KUKA KRL program: f1_Kuka_APT221T03S21.SRC

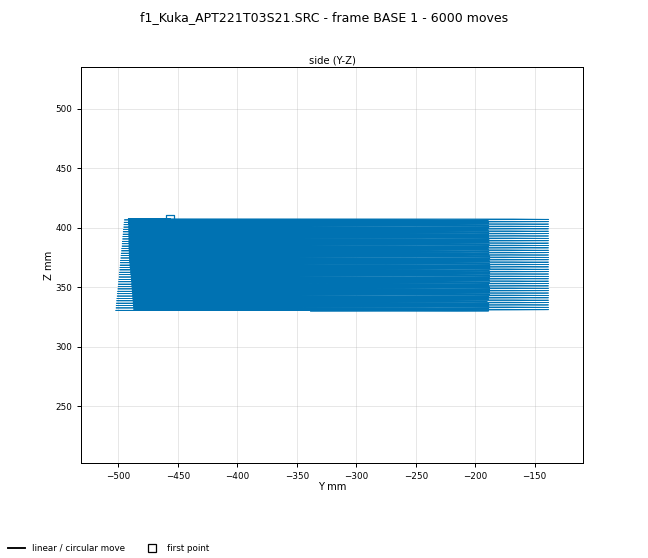
[picture p0: tool path of f1_Kuka_APT221T03S21.SRC in frame BASE 1, 6000 of 6001 moves have a stored position in this frame; points joined in program order, loops and branches not executed]
&ACCESS RVP
&REL 2
&PARAM TEMPLATE = C:\KRC\Roboter\Template\vorgabe
&PARAM EDITMASK = *
DEF f1_Kuka_APT221T03S21()


;FOLD INI;%{PE}%V3.2.0,%MKUKATPBASIS,%CINIT,%VCOMMON,%P
  ;FOLD BAS INI;%{E}%V3.2.0,%MKUKATPBASIS,%CINIT,%VINIT,%P
    GLOBAL INTERRUPT DECL 3 WHEN $STOPMESS==TRUE DO IR_STOPM ( )
    INTERRUPT ON 3
    BAS (#INITMOV,0 )
  ;ENDFOLD (BAS INI)
  ;FOLD USER INI;%{E}%V3.2.0,%MKUKATPUSER,%CINIT,%VINIT,%P
    ;Make your modifications here
  ;ENDFOLD (USER INI)
;ENDFOLD (INI)


;*** Make Null PTP Move
  PTP $pos_act

;*** Auto Load The Correct TOOL Data
  $tool=tool_data[3]

;*** Auto Load The Correct BASE Data
  $base=base_data[1]

  $ADVANCE = 5

;*** Restate Last Velocity
MMPM(30000.0)
SetRPM(6000)
LIN {X 0.057,Y -456.477,Z 407.554,A 0.000,B 0.000,C 90.000,E1 279.792} C_DIS
LIN {X 0.170,Y -464.178,Z 407.549,A 0.000,B 0.000,C 90.000,E1 278.746} C_DIS
LIN {X -0.091,Y -471.149,Z 407.543,A 0.000,B 0.000,C 90.000,E1 277.757} C_DIS
LIN {X 0.127,Y -477.448,Z 407.537,A 0.000,B 0.000,C 90.000,E1 276.720} C_DIS
LIN {X 0.133,Y -481.722,Z 407.533,A 0.000,B 0.000,C 90.000,E1 275.967} C_DIS
LIN {X 0.120,Y -485.329,Z 407.529,A 0.000,B 0.000,C 90.000,E1 275.220} C_DIS
LIN {X -0.179,Y -487.279,Z 407.526,A 0.000,B 0.000,C 90.000,E1 274.759} C_DIS
LIN {X -0.024,Y -488.832,Z 407.524,A 0.000,B 0.000,C 90.000,E1 274.245} C_DIS
LIN {X 0.180,Y -490.093,Z 407.521,A 0.000,B 0.000,C 90.000,E1 273.726} C_DIS
LIN {X -0.127,Y -490.997,Z 407.518,A 0.000,B 0.000,C 90.000,E1 273.269} C_DIS
LIN {X 0.090,Y -491.586,Z 407.515,A 0.000,B 0.000,C 90.000,E1 272.751} C_DIS
LIN {X -0.203,Y -491.810,Z 407.513,A 0.000,B 0.000,C 90.000,E1 272.293} C_DIS
LIN {X 0.017,Y -491.755,Z 407.510,A 0.000,B 0.000,C 90.000,E1 271.776} C_DIS
LIN {X 0.220,Y -491.256,Z 407.507,A 0.000,B 0.000,C 90.000,E1 271.260} C_DIS
LIN {X -0.065,Y -490.343,Z 407.504,A 0.000,B 0.000,C 90.000,E1 270.802} C_DIS
LIN {X 0.137,Y -488.944,Z 407.502,A 0.000,B 0.000,C 90.000,E1 270.286} C_DIS
LIN {X -0.154,Y -487.031,Z 407.499,A 0.000,B 0.000,C 90.000,E1 269.828} C_DIS
LIN {X 0.035,Y -484.413,Z 407.496,A 0.000,B 0.000,C 90.000,E1 269.312} C_DIS
LIN {X -0.123,Y -482.874,Z 407.495,A 0.000,B 0.000,C 90.000,E1 269.083} C_DIS
LIN {X 0.037,Y -479.075,Z 407.492,A 0.000,B 0.000,C 90.000,E1 268.568} C_DIS
LIN {X 0.188,Y -474.250,Z 407.489,A 0.000,B 0.000,C 90.000,E1 268.051} C_DIS
LIN {X 0.015,Y -471.372,Z 407.488,A 0.000,B 0.000,C 90.000,E1 267.822} C_DIS
LIN {X 0.040,Y -468.431,Z 407.487,A 0.000,B 0.000,C 90.000,E1 267.593} C_DIS
LIN {X 0.066,Y -465.066,Z 407.485,A 0.000,B 0.000,C 90.000,E1 267.364} C_DIS
LIN {X -0.070,Y -461.868,Z 407.484,A 0.000,B 0.000,C 90.000,E1 267.192} C_DIS
LIN {X -0.016,Y -454.836,Z 407.482,A 0.000,B 0.000,C 90.000,E1 266.846} C_DIS
LIN {X 0.077,Y -447.757,Z 407.481,A 0.000,B 0.000,C 90.000,E1 266.560} C_DIS
LIN {X 0.114,Y -440.498,Z 407.480,A 0.000,B 0.000,C 90.000,E1 266.331} C_DIS
LIN {X 0.063,Y -432.659,Z 407.479,A 0.000,B 0.000,C 90.000,E1 266.159} C_DIS
LIN {X -0.063,Y -423.683,Z 407.478,A 0.000,B 0.000,C 90.000,E1 266.045} C_DIS
LIN {X -0.172,Y -414.716,Z 407.478,A 0.000,B 0.000,C 90.000,E1 265.988} C_DIS
LIN {X 0.134,Y -409.225,Z 407.477,A 0.000,B 0.000,C 90.000,E1 265.927} C_DIS
LIN {X 0.029,Y -180.918,Z 407.477,A 0.000,B 0.000,C 90.000,E1 265.927} C_DIS
LIN {X 0.004,Y -180.835,Z 407.472,A 0.000,B 0.000,C 90.000,E1 264.894} C_DIS
LIN {X 0.078,Y -178.874,Z 407.443,A 0.000,B 0.000,C 90.000,E1 259.634} C_DIS
LIN {X -0.022,Y -175.916,Z 407.414,A 0.000,B 0.000,C 90.000,E1 254.574} C_DIS
LIN {X 0.034,Y -174.609,Z 407.405,A 0.000,B 0.000,C 90.000,E1 252.851} C_DIS
LIN {X -0.040,Y -171.590,Z 407.381,A 0.000,B 0.000,C 90.000,E1 248.592} C_DIS
LIN {X -0.050,Y -167.813,Z 407.357,A 0.000,B 0.000,C 90.000,E1 244.280} C_DIS
LIN {X -0.033,Y -166.534,Z 407.347,A 0.000,B 0.000,C 90.000,E1 242.538} C_DIS
LIN {X 0.017,Y -162.533,Z 407.323,A 0.000,B 0.000,C 90.000,E1 238.152} C_DIS
LIN {X -0.061,Y -161.208,Z 407.313,A 0.000,B 0.000,C 90.000,E1 236.421} C_DIS
LIN {X -0.026,Y -157.216,Z 407.289,A 0.000,B 0.000,C 90.000,E1 231.984} C_DIS
LIN {X -0.002,Y -155.943,Z 407.279,A 0.000,B 0.000,C 90.000,E1 230.194} C_DIS
LIN {X -0.043,Y -152.196,Z 407.254,A 0.000,B 0.000,C 90.000,E1 225.729} C_DIS
LIN {X -0.022,Y -150.442,Z 407.239,A 0.000,B 0.000,C 90.000,E1 223.014} C_DIS
LIN {X 0.005,Y -147.168,Z 407.214,A 0.000,B 0.000,C 90.000,E1 218.463} C_DIS
LIN {X -0.028,Y -145.184,Z 407.193,A 0.000,B 0.000,C 90.000,E1 214.818} C_DIS
LIN {X 0.008,Y -142.329,Z 407.163,A 0.000,B 0.000,C 90.000,E1 209.283} C_DIS
LIN {X 0.002,Y -141.717,Z 407.152,A 0.000,B 0.000,C 90.000,E1 207.436} C_DIS
LIN {X 0.050,Y -139.475,Z 407.116,A 0.000,B 0.000,C 90.000,E1 200.918} C_DIS
LIN {X 0.041,Y -138.972,Z 407.101,A 0.000,B 0.000,C 90.000,E1 198.127} C_DIS
LIN {X 0.030,Y -138.330,Z 407.054,A 0.000,B 0.000,C 90.000,E1 189.726} C_DIS
LIN {X 0.033,Y -139.435,Z 407.007,A 0.000,B 0.000,C 90.000,E1 181.318} C_DIS
LIN {X -0.027,Y -140.965,Z 406.976,A 0.000,B 0.000,C 90.000,E1 175.755} C_DIS
LIN {X 0.064,Y -142.720,Z 406.956,A 0.000,B 0.000,C 90.000,E1 172.008} C_DIS
LIN {X 0.022,Y -145.101,Z 406.930,A 0.000,B 0.000,C 90.000,E1 167.409} C_DIS
LIN {X 0.017,Y -147.725,Z 406.910,A 0.000,B 0.000,C 90.000,E1 163.740} C_DIS
LIN {X -0.042,Y -150.386,Z 406.889,A 0.000,B 0.000,C 90.000,E1 160.115} C_DIS
LIN {X -0.025,Y -153.817,Z 406.869,A 0.000,B 0.000,C 90.000,E1 156.485} C_DIS
LIN {X 0.035,Y -157.229,Z 406.849,A 0.000,B 0.000,C 90.000,E1 152.871} C_DIS
LIN {X -0.024,Y -161.397,Z 406.830,A 0.000,B 0.000,C 90.000,E1 149.331} C_DIS
LIN {X -0.014,Y -165.599,Z 406.810,A 0.000,B 0.000,C 90.000,E1 145.801} C_DIS
LIN {X -0.028,Y -170.523,Z 406.791,A 0.000,B 0.000,C 90.000,E1 142.316} C_DIS
LIN {X 0.015,Y -175.403,Z 406.771,A 0.000,B 0.000,C 90.000,E1 138.852} C_DIS
LIN {X 0.006,Y -181.026,Z 406.752,A 0.000,B 0.000,C 90.000,E1 135.445} C_DIS
LIN {X 0.000,Y -186.458,Z 406.734,A 0.000,B 0.000,C 90.000,E1 132.081} C_DIS
LIN {X 0.068,Y -191.082,Z 406.720,A 0.000,B 0.000,C 90.000,E1 129.564} C_DIS
LIN {X -0.005,Y -197.267,Z 406.701,A 0.000,B 0.000,C 90.000,E1 126.091} C_DIS
LIN {X -0.043,Y -296.085,Z 406.700,A 0.000,B 0.000,C 90.000,E1 126.091} C_DIS
LIN {X 0.068,Y -298.942,Z 406.700,A 0.000,B 0.000,C 90.000,E1 126.011} C_DIS
LIN {X 0.142,Y -303.617,Z 406.699,A 0.000,B 0.000,C 90.000,E1 125.724} C_DIS
LIN {X 0.039,Y -306.311,Z 406.697,A 0.000,B 0.000,C 90.000,E1 125.471} C_DIS
LIN {X 0.054,Y -310.021,Z 406.694,A 0.000,B 0.000,C 90.000,E1 124.898} C_DIS
LIN {X -0.167,Y -311.511,Z 406.692,A 0.000,B 0.000,C 90.000,E1 124.612} C_DIS
LIN {X 0.005,Y -316.928,Z 406.683,A 0.000,B 0.000,C 90.000,E1 122.959} C_DIS
LIN {X 0.033,Y -327.394,Z 406.667,A 0.000,B 0.000,C 90.000,E1 120.079} C_DIS
LIN {X 0.034,Y -339.228,Z 406.651,A 0.000,B 0.000,C 90.000,E1 117.257} C_DIS
LIN {X -0.100,Y -352.532,Z 406.636,A 0.000,B 0.000,C 90.000,E1 114.515} C_DIS
LIN {X 0.102,Y -365.691,Z 406.623,A 0.000,B 0.000,C 90.000,E1 112.078} C_DIS
LIN {X -0.112,Y -380.206,Z 406.610,A 0.000,B 0.000,C 90.000,E1 109.758} C_DIS
LIN {X -0.094,Y -396.183,Z 406.597,A 0.000,B 0.000,C 90.000,E1 107.457} C_DIS
LIN {X 0.091,Y -413.738,Z 406.584,A 0.000,B 0.000,C 90.000,E1 105.190} C_DIS
LIN {X 0.132,Y -432.973,Z 406.572,A 0.000,B 0.000,C 90.000,E1 103.008} C_DIS
LIN {X -0.111,Y -453.179,Z 406.561,A 0.000,B 0.000,C 90.000,E1 101.007} C_DIS
LIN {X -0.181,Y -473.926,Z 406.551,A 0.000,B 0.000,C 90.000,E1 99.151} C_DIS
LIN {X -0.056,Y -487.135,Z 406.545,A 0.000,B 0.000,C 90.000,E1 98.049} C_DIS
LIN {X -0.228,Y -490.973,Z 406.542,A 0.000,B 0.000,C 90.000,E1 97.644} C_DIS
LIN {X 0.151,Y -492.454,Z 406.541,A 0.000,B 0.000,C 90.000,E1 97.352} C_DIS
LIN {X -0.020,Y -493.557,Z 406.540,A 0.000,B 0.000,C 90.000,E1 97.125} C_DIS
LIN {X 0.220,Y -494.847,Z 406.537,A 0.000,B 0.000,C 90.000,E1 96.606} C_DIS
LIN {X -0.024,Y -495.105,Z 406.534,A 0.000,B 0.000,C 90.000,E1 96.144} C_DIS
LIN {X 0.229,Y -494.370,Z 406.531,A 0.000,B 0.000,C 90.000,E1 95.625} C_DIS
LIN {X -0.009,Y -492.516,Z 406.529,A 0.000,B 0.000,C 90.000,E1 95.163} C_DIS
LIN {X -0.152,Y -491.055,Z 406.527,A 0.000,B 0.000,C 90.000,E1 94.935} C_DIS
LIN {X -0.186,Y -483.507,Z 406.522,A 0.000,B 0.000,C 90.000,E1 93.955} C_DIS
LIN {X -0.221,Y -471.556,Z 406.514,A 0.000,B 0.000,C 90.000,E1 92.465} C_DIS
LIN {X -0.182,Y -454.336,Z 406.501,A 0.000,B 0.000,C 90.000,E1 90.172} C_DIS
LIN {X -0.062,Y -433.473,Z 406.483,A 0.000,B 0.000,C 90.000,E1 87.020} C_DIS
LIN {X 0.062,Y -417.355,Z 406.468,A 0.000,B 0.000,C 90.000,E1 84.318} C_DIS
LIN {X -0.032,Y -406.574,Z 406.458,A 0.000,B 0.000,C 90.000,E1 82.413} C_DIS
LIN {X -0.130,Y -392.920,Z 406.444,A 0.000,B 0.000,C 90.000,E1 79.916} C_DIS
LIN {X -0.171,Y -381.020,Z 406.431,A 0.000,B 0.000,C 90.000,E1 77.645} C_DIS
LIN {X 0.109,Y -369.476,Z 406.418,A 0.000,B 0.000,C 90.000,E1 75.283} C_DIS
LIN {X -0.142,Y -355.454,Z 406.402,A 0.000,B 0.000,C 90.000,E1 72.362} C_DIS
LIN {X -0.047,Y -343.515,Z 406.387,A 0.000,B 0.000,C 90.000,E1 69.625} C_DIS
LIN {X -0.146,Y -333.190,Z 406.373,A 0.000,B 0.000,C 90.000,E1 67.177} C_DIS
LIN {X -0.116,Y -323.180,Z 406.359,A 0.000,B 0.000,C 90.000,E1 64.665} C_DIS
LIN {X 0.012,Y -312.410,Z 406.343,A 0.000,B 0.000,C 90.000,E1 61.769} C_DIS
LIN {X -0.105,Y -301.020,Z 406.325,A 0.000,B 0.000,C 90.000,E1 58.535} C_DIS
LIN {X 0.085,Y -290.585,Z 406.307,A 0.000,B 0.000,C 90.000,E1 55.182} C_DIS
LIN {X -0.015,Y -280.969,Z 406.288,A 0.000,B 0.000,C 90.000,E1 51.823} C_DIS
LIN {X 0.086,Y -275.411,Z 406.276,A 0.000,B 0.000,C 90.000,E1 49.747} C_DIS
LIN {X 0.052,Y -269.718,Z 406.265,A 0.000,B 0.000,C 90.000,E1 47.676} C_DIS
LIN {X 0.091,Y -263.780,Z 406.253,A 0.000,B 0.000,C 90.000,E1 45.567} C_DIS
LIN {X 0.010,Y -257.732,Z 406.241,A 0.000,B 0.000,C 90.000,E1 43.461} C_DIS
LIN {X 0.017,Y -251.549,Z 406.230,A 0.000,B 0.000,C 90.000,E1 41.310} C_DIS
LIN {X 0.105,Y -243.317,Z 406.213,A 0.000,B 0.000,C 90.000,E1 38.382} C_DIS
LIN {X 0.060,Y -233.444,Z 406.193,A 0.000,B 0.000,C 90.000,E1 34.692} C_DIS
LIN {X 0.083,Y -226.277,Z 406.176,A 0.000,B 0.000,C 90.000,E1 31.671} C_DIS
LIN {X 0.060,Y -218.050,Z 406.155,A 0.000,B 0.000,C 90.000,E1 27.847} C_DIS
LIN {X -0.076,Y -212.245,Z 406.138,A 0.000,B 0.000,C 90.000,E1 24.771} C_DIS
LIN {X 0.063,Y -205.875,Z 406.116,A 0.000,B 0.000,C 90.000,E1 20.791} C_DIS
LIN {X 0.031,Y -200.411,Z 406.093,A 0.000,B 0.000,C 90.000,E1 16.804} C_DIS
LIN {X -0.002,Y -195.980,Z 406.071,A 0.000,B 0.000,C 90.000,E1 12.771} C_DIS
LIN {X 0.032,Y -192.503,Z 406.048,A 0.000,B 0.000,C 90.000,E1 8.681} C_DIS
LIN {X 0.027,Y -189.559,Z 406.016,A 0.000,B 0.000,C 90.000,E1 2.922} C_DIS
LIN {X -0.068,Y -189.023,Z 405.974,A 0.000,B 0.000,C 90.000,E1 355.412} C_DIS
LIN {X 0.078,Y -191.530,Z 405.938,A 0.000,B 0.000,C 90.000,E1 348.757} C_DIS
LIN {X -0.046,Y -194.931,Z 405.910,A 0.000,B 0.000,C 90.000,E1 343.866} C_DIS
LIN {X 0.082,Y -198.897,Z 405.888,A 0.000,B 0.000,C 90.000,E1 339.752} C_DIS
LIN {X -0.013,Y -203.955,Z 405.865,A 0.000,B 0.000,C 90.000,E1 335.741} C_DIS
LIN {X -0.089,Y -210.064,Z 405.843,A 0.000,B 0.000,C 90.000,E1 331.769} C_DIS
LIN {X 0.069,Y -216.918,Z 405.821,A 0.000,B 0.000,C 90.000,E1 327.788} C_DIS
LIN {X 0.064,Y -224.337,Z 405.800,A 0.000,B 0.000,C 90.000,E1 323.909} C_DIS
LIN {X -0.029,Y -232.586,Z 405.778,A 0.000,B 0.000,C 90.000,E1 320.114} C_DIS
LIN {X -0.032,Y -239.931,Z 405.762,A 0.000,B 0.000,C 90.000,E1 317.106} C_DIS
LIN {X -0.051,Y -249.284,Z 405.743,A 0.000,B 0.000,C 90.000,E1 313.785} C_DIS
LIN {X -0.119,Y -259.993,Z 405.725,A 0.000,B 0.000,C 90.000,E1 310.539} C_DIS
LIN {X 0.034,Y -271.763,Z 405.707,A 0.000,B 0.000,C 90.000,E1 307.317} C_DIS
LIN {X -0.002,Y -285.718,Z 405.688,A 0.000,B 0.000,C 90.000,E1 303.865} C_DIS
LIN {X 0.171,Y -300.414,Z 405.669,A 0.000,B 0.000,C 90.000,E1 300.463} C_DIS
LIN {X 0.053,Y -311.660,Z 405.657,A 0.000,B 0.000,C 90.000,E1 298.180} C_DIS
LIN {X 0.074,Y -327.714,Z 405.641,A 0.000,B 0.000,C 90.000,E1 295.283} C_DIS
LIN {X 0.151,Y -339.486,Z 405.630,A 0.000,B 0.000,C 90.000,E1 293.387} C_DIS
LIN {X -0.044,Y -358.914,Z 405.615,A 0.000,B 0.000,C 90.000,E1 290.663} C_DIS
LIN {X 0.048,Y -379.551,Z 405.600,A 0.000,B 0.000,C 90.000,E1 288.000} C_DIS
LIN {X 0.190,Y -404.938,Z 405.585,A 0.000,B 0.000,C 90.000,E1 285.190} C_DIS
LIN {X -0.153,Y -422.776,Z 405.575,A 0.000,B 0.000,C 90.000,E1 283.467} C_DIS
LIN {X 0.019,Y -435.520,Z 405.568,A 0.000,B 0.000,C 90.000,E1 282.175} C_DIS
LIN {X -0.089,Y -442.879,Z 405.563,A 0.000,B 0.000,C 90.000,E1 281.422} C_DIS
LIN {X 0.147,Y -449.870,Z 405.559,A 0.000,B 0.000,C 90.000,E1 280.602} C_DIS
LIN {X -0.085,Y -456.195,Z 405.555,A 0.000,B 0.000,C 90.000,E1 279.849} C_DIS
LIN {X -0.185,Y -462.061,Z 405.550,A 0.000,B 0.000,C 90.000,E1 279.086} C_DIS
LIN {X -0.083,Y -469.205,Z 405.545,A 0.000,B 0.000,C 90.000,E1 278.049} C_DIS
LIN {X 0.114,Y -475.706,Z 405.539,A 0.000,B 0.000,C 90.000,E1 277.011} C_DIS
LIN {X 0.103,Y -480.119,Z 405.535,A 0.000,B 0.000,C 90.000,E1 276.258} C_DIS
LIN {X 0.083,Y -483.997,Z 405.531,A 0.000,B 0.000,C 90.000,E1 275.511} C_DIS
LIN {X 0.136,Y -487.131,Z 405.527,A 0.000,B 0.000,C 90.000,E1 274.759} C_DIS
LIN {X -0.198,Y -488.697,Z 405.524,A 0.000,B 0.000,C 90.000,E1 274.302} C_DIS
LIN {X 0.005,Y -489.926,Z 405.521,A 0.000,B 0.000,C 90.000,E1 273.784} C_DIS
LIN {X 0.187,Y -490.846,Z 405.518,A 0.000,B 0.000,C 90.000,E1 273.269} C_DIS
LIN {X -0.088,Y -491.442,Z 405.516,A 0.000,B 0.000,C 90.000,E1 272.808} C_DIS
LIN {X 0.109,Y -491.707,Z 405.513,A 0.000,B 0.000,C 90.000,E1 272.293} C_DIS
LIN {X -0.179,Y -491.638,Z 405.510,A 0.000,B 0.000,C 90.000,E1 271.835} C_DIS
LIN {X 0.040,Y -491.251,Z 405.507,A 0.000,B 0.000,C 90.000,E1 271.318} C_DIS
LIN {X 0.244,Y -490.356,Z 405.505,A 0.000,B 0.000,C 90.000,E1 270.802} C_DIS
LIN {X -0.044,Y -489.016,Z 405.502,A 0.000,B 0.000,C 90.000,E1 270.344} C_DIS
LIN {X 0.153,Y -487.140,Z 405.499,A 0.000,B 0.000,C 90.000,E1 269.828} C_DIS
LIN {X -0.143,Y -484.631,Z 405.496,A 0.000,B 0.000,C 90.000,E1 269.370} C_DIS
LIN {X 0.027,Y -481.322,Z 405.494,A 0.000,B 0.000,C 90.000,E1 268.854} C_DIS
LIN {X -0.138,Y -479.424,Z 405.492,A 0.000,B 0.000,C 90.000,E1 268.625} C_DIS
LIN {X 0.017,Y -474.712,Z 405.490,A 0.000,B 0.000,C 90.000,E1 268.108} C_DIS
LIN {X -0.127,Y -468.991,Z 405.487,A 0.000,B 0.000,C 90.000,E1 267.650} C_DIS
LIN {X 0.208,Y -462.514,Z 405.485,A 0.000,B 0.000,C 90.000,E1 267.192} C_DIS
LIN {X 0.180,Y -455.557,Z 405.483,A 0.000,B 0.000,C 90.000,E1 266.849} C_DIS
LIN {X -0.214,Y -448.411,Z 405.481,A 0.000,B 0.000,C 90.000,E1 266.617} C_DIS
LIN {X -0.214,Y -441.149,Z 405.480,A 0.000,B 0.000,C 90.000,E1 266.388} C_DIS
LIN {X 0.140,Y -433.393,Z 405.479,A 0.000,B 0.000,C 90.000,E1 266.159} C_DIS
LIN {X -0.020,Y -424.376,Z 405.478,A 0.000,B 0.000,C 90.000,E1 266.045} C_DIS
LIN {X -0.152,Y -416.010,Z 405.478,A 0.000,B 0.000,C 90.000,E1 265.988} C_DIS
LIN {X 0.123,Y -411.862,Z 405.477,A 0.000,B 0.000,C 90.000,E1 265.931} C_DIS
LIN {X 0.037,Y -180.917,Z 405.477,A 0.000,B 0.000,C 90.000,E1 265.927} C_DIS
LIN {X 0.009,Y -180.835,Z 405.472,A 0.000,B 0.000,C 90.000,E1 264.894} C_DIS
LIN {X -0.094,Y -178.874,Z 405.443,A 0.000,B 0.000,C 90.000,E1 259.690} C_DIS
LIN {X -0.017,Y -175.917,Z 405.414,A 0.000,B 0.000,C 90.000,E1 254.574} C_DIS
LIN {X 0.039,Y -174.610,Z 405.405,A 0.000,B 0.000,C 90.000,E1 252.851} C_DIS
LIN {X -0.035,Y -171.592,Z 405.381,A 0.000,B 0.000,C 90.000,E1 248.592} C_DIS
LIN {X -0.046,Y -167.814,Z 405.357,A 0.000,B 0.000,C 90.000,E1 244.280} C_DIS
LIN {X -0.029,Y -166.536,Z 405.347,A 0.000,B 0.000,C 90.000,E1 242.538} C_DIS
LIN {X 0.021,Y -162.534,Z 405.323,A 0.000,B 0.000,C 90.000,E1 238.152} C_DIS
LIN {X -0.057,Y -161.209,Z 405.313,A 0.000,B 0.000,C 90.000,E1 236.421} C_DIS
LIN {X -0.021,Y -157.218,Z 405.289,A 0.000,B 0.000,C 90.000,E1 231.984} C_DIS
LIN {X 0.002,Y -155.944,Z 405.279,A 0.000,B 0.000,C 90.000,E1 230.194} C_DIS
LIN {X -0.038,Y -152.197,Z 405.254,A 0.000,B 0.000,C 90.000,E1 225.729} C_DIS
LIN {X -0.017,Y -150.443,Z 405.239,A 0.000,B 0.000,C 90.000,E1 223.014} C_DIS
LIN {X 0.010,Y -147.169,Z 405.214,A 0.000,B 0.000,C 90.000,E1 218.463} C_DIS
LIN {X -0.023,Y -145.185,Z 405.193,A 0.000,B 0.000,C 90.000,E1 214.818} C_DIS
LIN {X 0.011,Y -142.329,Z 405.163,A 0.000,B 0.000,C 90.000,E1 209.283} C_DIS
LIN {X 0.006,Y -141.718,Z 405.152,A 0.000,B 0.000,C 90.000,E1 207.436} C_DIS
LIN {X 0.054,Y -139.476,Z 405.116,A 0.000,B 0.000,C 90.000,E1 200.918} C_DIS
LIN {X 0.045,Y -138.972,Z 405.101,A 0.000,B 0.000,C 90.000,E1 198.127} C_DIS
LIN {X 0.035,Y -138.330,Z 405.054,A 0.000,B 0.000,C 90.000,E1 189.726} C_DIS
LIN {X 0.037,Y -139.435,Z 405.007,A 0.000,B 0.000,C 90.000,E1 181.318} C_DIS
LIN {X -0.023,Y -140.963,Z 404.976,A 0.000,B 0.000,C 90.000,E1 175.755} C_DIS
LIN {X 0.068,Y -142.720,Z 404.956,A 0.000,B 0.000,C 90.000,E1 172.008} C_DIS
LIN {X 0.026,Y -145.100,Z 404.930,A 0.000,B 0.000,C 90.000,E1 167.409} C_DIS
LIN {X 0.022,Y -147.724,Z 404.910,A 0.000,B 0.000,C 90.000,E1 163.740} C_DIS
LIN {X -0.038,Y -150.384,Z 404.889,A 0.000,B 0.000,C 90.000,E1 160.115} C_DIS
LIN {X -0.020,Y -153.816,Z 404.869,A 0.000,B 0.000,C 90.000,E1 156.485} C_DIS
LIN {X 0.038,Y -157.227,Z 404.849,A 0.000,B 0.000,C 90.000,E1 152.871} C_DIS
LIN {X -0.020,Y -161.395,Z 404.830,A 0.000,B 0.000,C 90.000,E1 149.331} C_DIS
LIN {X -0.010,Y -165.596,Z 404.810,A 0.000,B 0.000,C 90.000,E1 145.801} C_DIS
LIN {X -0.024,Y -170.520,Z 404.791,A 0.000,B 0.000,C 90.000,E1 142.316} C_DIS
LIN {X 0.020,Y -175.400,Z 404.771,A 0.000,B 0.000,C 90.000,E1 138.852} C_DIS
LIN {X 0.011,Y -181.024,Z 404.753,A 0.000,B 0.000,C 90.000,E1 135.445} C_DIS
LIN {X 0.005,Y -186.456,Z 404.734,A 0.000,B 0.000,C 90.000,E1 132.081} C_DIS
LIN {X 0.074,Y -191.080,Z 404.720,A 0.000,B 0.000,C 90.000,E1 129.564} C_DIS
LIN {X -0.096,Y -197.318,Z 404.700,A 0.000,B 0.000,C 90.000,E1 126.091} C_DIS
LIN {X 0.081,Y -197.374,Z 404.700,A 0.000,B 0.000,C 90.000,E1 126.011} C_DIS
LIN {X 0.072,Y -296.560,Z 404.700,A 0.000,B 0.000,C 90.000,E1 126.011} C_DIS
LIN {X 0.021,Y -300.932,Z 404.699,A 0.000,B 0.000,C 90.000,E1 125.884} C_DIS
LIN {X 0.148,Y -303.059,Z 404.699,A 0.000,B 0.000,C 90.000,E1 125.724} C_DIS
LIN {X 0.046,Y -305.973,Z 404.697,A 0.000,B 0.000,C 90.000,E1 125.471} C_DIS
LIN {X -0.005,Y -309.689,Z 404.694,A 0.000,B 0.000,C 90.000,E1 124.945} C_DIS
LIN {X 0.027,Y -311.284,Z 404.692,A 0.000,B 0.000,C 90.000,E1 124.612} C_DIS
LIN {X -0.147,Y -313.589,Z 404.689,A 0.000,B 0.000,C 90.000,E1 123.992} C_DIS
LIN {X 0.113,Y -323.609,Z 404.673,A 0.000,B 0.000,C 90.000,E1 121.052} C_DIS
LIN {X 0.003,Y -334.956,Z 404.657,A 0.000,B 0.000,C 90.000,E1 118.231} C_DIS
LIN {X -0.104,Y -347.741,Z 404.641,A 0.000,B 0.000,C 90.000,E1 115.463} C_DIS
LIN {X -0.023,Y -360.401,Z 404.628,A 0.000,B 0.000,C 90.000,E1 113.025} C_DIS
LIN {X -0.098,Y -374.378,Z 404.615,A 0.000,B 0.000,C 90.000,E1 110.663} C_DIS
LIN {X 0.139,Y -389.774,Z 404.602,A 0.000,B 0.000,C 90.000,E1 108.308} C_DIS
LIN {X -0.099,Y -406.702,Z 404.589,A 0.000,B 0.000,C 90.000,E1 106.079} C_DIS
LIN {X -0.168,Y -425.287,Z 404.577,A 0.000,B 0.000,C 90.000,E1 103.883} C_DIS
LIN {X -0.087,Y -445.249,Z 404.565,A 0.000,B 0.000,C 90.000,E1 101.771} C_DIS
LIN {X -0.130,Y -465.793,Z 404.555,A 0.000,B 0.000,C 90.000,E1 99.849} C_DIS
LIN {X 0.135,Y -486.836,Z 404.545,A 0.000,B 0.000,C 90.000,E1 98.049} C_DIS
LIN {X -0.133,Y -489.109,Z 404.544,A 0.000,B 0.000,C 90.000,E1 97.871} C_DIS
LIN {X 0.017,Y -490.838,Z 404.542,A 0.000,B 0.000,C 90.000,E1 97.644} C_DIS
LIN {X -0.085,Y -492.396,Z 404.541,A 0.000,B 0.000,C 90.000,E1 97.409} C_DIS
LIN {X -0.253,Y -493.561,Z 404.540,A 0.000,B 0.000,C 90.000,E1 97.182} C_DIS
LIN {X -0.013,Y -494.956,Z 404.537,A 0.000,B 0.000,C 90.000,E1 96.663} C_DIS
LIN {X 0.234,Y -495.305,Z 404.534,A 0.000,B 0.000,C 90.000,E1 96.144} C_DIS
LIN {X -0.005,Y -494.663,Z 404.532,A 0.000,B 0.000,C 90.000,E1 95.682} C_DIS
LIN {X 0.249,Y -492.924,Z 404.529,A 0.000,B 0.000,C 90.000,E1 95.163} C_DIS
LIN {X 0.108,Y -491.539,Z 404.527,A 0.000,B 0.000,C 90.000,E1 94.935} C_DIS
LIN {X 0.075,Y -484.085,Z 404.522,A 0.000,B 0.000,C 90.000,E1 93.955} C_DIS
LIN {X 0.041,Y -472.141,Z 404.514,A 0.000,B 0.000,C 90.000,E1 92.465} C_DIS
LIN {X 0.086,Y -454.883,Z 404.501,A 0.000,B 0.000,C 90.000,E1 90.172} C_DIS
LIN {X 0.047,Y -435.606,Z 404.485,A 0.000,B 0.000,C 90.000,E1 87.306} C_DIS
LIN {X -0.077,Y -417.802,Z 404.469,A 0.000,B 0.000,C 90.000,E1 84.375} C_DIS
LIN {X -0.158,Y -407.017,Z 404.458,A 0.000,B 0.000,C 90.000,E1 82.470} C_DIS
LIN {X 0.082,Y -393.372,Z 404.444,A 0.000,B 0.000,C 90.000,E1 79.926} C_DIS
LIN {X 0.112,Y -381.495,Z 404.431,A 0.000,B 0.000,C 90.000,E1 77.645} C_DIS
LIN {X 0.028,Y -368.482,Z 404.417,A 0.000,B 0.000,C 90.000,E1 75.046} C_DIS
LIN {X 0.085,Y -354.496,Z 404.400,A 0.000,B 0.000,C 90.000,E1 72.072} C_DIS
LIN {X -0.182,Y -342.545,Z 404.385,A 0.000,B 0.000,C 90.000,E1 69.390} C_DIS
LIN {X -0.178,Y -332.212,Z 404.372,A 0.000,B 0.000,C 90.000,E1 66.922} C_DIS
LIN {X -0.168,Y -322.194,Z 404.358,A 0.000,B 0.000,C 90.000,E1 64.409} C_DIS
LIN {X -0.069,Y -311.468,Z 404.342,A 0.000,B 0.000,C 90.000,E1 61.513} C_DIS
LIN {X -0.033,Y -299.051,Z 404.322,A 0.000,B 0.000,C 90.000,E1 57.916} C_DIS
LIN {X 0.095,Y -288.784,Z 404.303,A 0.000,B 0.000,C 90.000,E1 54.562} C_DIS
LIN {X 0.106,Y -279.308,Z 404.284,A 0.000,B 0.000,C 90.000,E1 51.170} C_DIS
LIN {X -0.048,Y -271.855,Z 404.269,A 0.000,B 0.000,C 90.000,E1 48.447} C_DIS
LIN {X -0.146,Y -265.998,Z 404.257,A 0.000,B 0.000,C 90.000,E1 46.377} C_DIS
LIN {X 0.001,Y -260.007,Z 404.246,A 0.000,B 0.000,C 90.000,E1 44.231} C_DIS
LIN {X 0.045,Y -253.893,Z 404.234,A 0.000,B 0.000,C 90.000,E1 42.081} C_DIS
LIN {X 0.005,Y -245.664,Z 404.218,A 0.000,B 0.000,C 90.000,E1 39.197} C_DIS
LIN {X 0.026,Y -237.629,Z 404.201,A 0.000,B 0.000,C 90.000,E1 36.251} C_DIS
LIN {X -0.099,Y -230.053,Z 404.185,A 0.000,B 0.000,C 90.000,E1 33.293} C_DIS
LIN {X 0.028,Y -221.491,Z 404.164,A 0.000,B 0.000,C 90.000,E1 29.461} C_DIS
LIN {X 0.070,Y -215.256,Z 404.147,A 0.000,B 0.000,C 90.000,E1 26.360} C_DIS
LIN {X -0.001,Y -208.502,Z 404.125,A 0.000,B 0.000,C 90.000,E1 22.461} C_DIS
LIN {X -0.008,Y -202.584,Z 404.103,A 0.000,B 0.000,C 90.000,E1 18.489} C_DIS
LIN {X -0.061,Y -197.713,Z 404.080,A 0.000,B 0.000,C 90.000,E1 14.481} C_DIS
LIN {X 0.107,Y -193.789,Z 404.058,A 0.000,B 0.000,C 90.000,E1 10.366} C_DIS
LIN {X -0.054,Y -190.984,Z 404.035,A 0.000,B 0.000,C 90.000,E1 6.315} C_DIS
LIN {X -0.034,Y -188.731,Z 403.997,A 0.000,B 0.000,C 90.000,E1 359.542} C_DIS
LIN {X -0.049,Y -190.574,Z 403.947,A 0.000,B 0.000,C 90.000,E1 350.443} C_DIS
LIN {X 0.083,Y -193.508,Z 403.919,A 0.000,B 0.000,C 90.000,E1 345.463} C_DIS
LIN {X -0.013,Y -197.032,Z 403.897,A 0.000,B 0.000,C 90.000,E1 341.402} C_DIS
LIN {X -0.057,Y -201.684,Z 403.874,A 0.000,B 0.000,C 90.000,E1 337.358} C_DIS
LIN {X -0.088,Y -206.142,Z 403.856,A 0.000,B 0.000,C 90.000,E1 334.152} C_DIS
LIN {X 0.103,Y -212.589,Z 403.834,A 0.000,B 0.000,C 90.000,E1 330.127} C_DIS
LIN {X 0.091,Y -219.685,Z 403.812,A 0.000,B 0.000,C 90.000,E1 326.215} C_DIS
LIN {X -0.063,Y -227.402,Z 403.791,A 0.000,B 0.000,C 90.000,E1 322.396} C_DIS
LIN {X -0.095,Y -236.048,Z 403.770,A 0.000,B 0.000,C 90.000,E1 318.609} C_DIS
LIN {X -0.053,Y -244.886,Z 403.751,A 0.000,B 0.000,C 90.000,E1 315.243} C_DIS
LIN {X 0.099,Y -254.970,Z 403.733,A 0.000,B 0.000,C 90.000,E1 311.919} C_DIS
LIN {X -0.136,Y -266.388,Z 403.715,A 0.000,B 0.000,C 90.000,E1 308.749} C_DIS
LIN {X -0.136,Y -278.513,Z 403.698,A 0.000,B 0.000,C 90.000,E1 305.598} C_DIS
LIN {X -0.007,Y -289.924,Z 403.682,A 0.000,B 0.000,C 90.000,E1 302.832} C_DIS
LIN {X -0.007,Y -305.022,Z 403.664,A 0.000,B 0.000,C 90.000,E1 299.489} C_DIS
LIN {X 0.070,Y -315.076,Z 403.653,A 0.000,B 0.000,C 90.000,E1 297.513} C_DIS
LIN {X -0.008,Y -327.730,Z 403.640,A 0.000,B 0.000,C 90.000,E1 295.283} C_DIS
LIN {X 0.051,Y -341.634,Z 403.628,A 0.000,B 0.000,C 90.000,E1 293.078} C_DIS
LIN {X -0.080,Y -361.268,Z 403.613,A 0.000,B 0.000,C 90.000,E1 290.355} C_DIS
LIN {X -0.025,Y -379.748,Z 403.600,A 0.000,B 0.000,C 90.000,E1 288.000} C_DIS
LIN {X 0.151,Y -405.137,Z 403.585,A 0.000,B 0.000,C 90.000,E1 285.190} C_DIS
LIN {X 0.140,Y -423.029,Z 403.575,A 0.000,B 0.000,C 90.000,E1 283.411} C_DIS
LIN {X -0.169,Y -435.849,Z 403.568,A 0.000,B 0.000,C 90.000,E1 282.175} C_DIS
LIN {X 0.109,Y -443.200,Z 403.563,A 0.000,B 0.000,C 90.000,E1 281.366} C_DIS
LIN {X -0.090,Y -450.175,Z 403.559,A 0.000,B 0.000,C 90.000,E1 280.602} C_DIS
LIN {X 0.127,Y -456.459,Z 403.555,A 0.000,B 0.000,C 90.000,E1 279.792} C_DIS
LIN {X -0.217,Y -464.128,Z 403.549,A 0.000,B 0.000,C 90.000,E1 278.803} C_DIS
LIN {X 0.142,Y -469.400,Z 403.544,A 0.000,B 0.000,C 90.000,E1 277.992} C_DIS
LIN {X -0.069,Y -475.887,Z 403.539,A 0.000,B 0.000,C 90.000,E1 277.004} C_DIS
LIN {X -0.137,Y -480.278,Z 403.535,A 0.000,B 0.000,C 90.000,E1 276.258} C_DIS
LIN {X -0.159,Y -484.142,Z 403.531,A 0.000,B 0.000,C 90.000,E1 275.511} C_DIS
LIN {X -0.107,Y -487.197,Z 403.526,A 0.000,B 0.000,C 90.000,E1 274.759} C_DIS
LIN {X 0.048,Y -488.730,Z 403.524,A 0.000,B 0.000,C 90.000,E1 274.245} C_DIS
LIN {X -0.237,Y -489.933,Z 403.521,A 0.000,B 0.000,C 90.000,E1 273.784} C_DIS
LIN {X -0.056,Y -490.798,Z 403.518,A 0.000,B 0.000,C 90.000,E1 273.269} C_DIS
LIN {X 0.160,Y -491.358,Z 403.515,A 0.000,B 0.000,C 90.000,E1 272.751} C_DIS
LIN {X -0.134,Y -491.616,Z 403.513,A 0.000,B 0.000,C 90.000,E1 272.293} C_DIS
LIN {X 0.085,Y -491.562,Z 403.510,A 0.000,B 0.000,C 90.000,E1 271.776} C_DIS
LIN {X -0.204,Y -491.099,Z 403.507,A 0.000,B 0.000,C 90.000,E1 271.318} C_DIS
LIN {X 0.000,Y -490.212,Z 403.504,A 0.000,B 0.000,C 90.000,E1 270.802} C_DIS
LIN {X 0.202,Y -488.877,Z 403.502,A 0.000,B 0.000,C 90.000,E1 270.286} C_DIS
LIN {X -0.090,Y -486.986,Z 403.499,A 0.000,B 0.000,C 90.000,E1 269.828} C_DIS
LIN {X 0.097,Y -484.465,Z 403.496,A 0.000,B 0.000,C 90.000,E1 269.312} C_DIS
LIN {X -0.217,Y -481.167,Z 403.493,A 0.000,B 0.000,C 90.000,E1 268.854} C_DIS
LIN {X 0.099,Y -479.190,Z 403.492,A 0.000,B 0.000,C 90.000,E1 268.568} C_DIS
LIN {X -0.224,Y -474.421,Z 403.489,A 0.000,B 0.000,C 90.000,E1 268.108} C_DIS
LIN {X 0.105,Y -468.633,Z 403.487,A 0.000,B 0.000,C 90.000,E1 267.593} C_DIS
LIN {X 0.132,Y -465.353,Z 403.485,A 0.000,B 0.000,C 90.000,E1 267.364} C_DIS
LIN {X -0.195,Y -458.304,Z 403.483,A 0.000,B 0.000,C 90.000,E1 267.020} C_DIS
LIN {X 0.146,Y -451.326,Z 403.482,A 0.000,B 0.000,C 90.000,E1 266.674} C_DIS
LIN {X 0.007,Y -444.134,Z 403.480,A 0.000,B 0.000,C 90.000,E1 266.445} C_DIS
LIN {X -0.220,Y -436.688,Z 403.479,A 0.000,B 0.000,C 90.000,E1 266.274} C_DIS
LIN {X -0.106,Y -428.385,Z 403.478,A 0.000,B 0.000,C 90.000,E1 266.102} C_DIS
LIN {X -0.209,Y -415.227,Z 403.478,A 0.000,B 0.000,C 90.000,E1 265.988} C_DIS
LIN {X 0.098,Y -409.742,Z 403.477,A 0.000,B 0.000,C 90.000,E1 265.927} C_DIS
LIN {X 0.014,Y -180.917,Z 403.477,A 0.000,B 0.000,C 90.000,E1 265.927} C_DIS
LIN {X -0.012,Y -180.834,Z 403.472,A 0.000,B 0.000,C 90.000,E1 264.894} C_DIS
LIN {X 0.061,Y -178.871,Z 403.443,A 0.000,B 0.000,C 90.000,E1 259.634} C_DIS
LIN {X -0.039,Y -175.914,Z 403.414,A 0.000,B 0.000,C 90.000,E1 254.574} C_DIS
LIN {X 0.018,Y -174.604,Z 403.405,A 0.000,B 0.000,C 90.000,E1 252.851} C_DIS
LIN {X -0.055,Y -171.587,Z 403.381,A 0.000,B 0.000,C 90.000,E1 248.592} C_DIS
LIN {X -0.066,Y -167.809,Z 403.357,A 0.000,B 0.000,C 90.000,E1 244.280} C_DIS
LIN {X -0.048,Y -166.530,Z 403.347,A 0.000,B 0.000,C 90.000,E1 242.538} C_DIS
LIN {X 0.087,Y -162.528,Z 403.323,A 0.000,B 0.000,C 90.000,E1 238.122} C_DIS
LIN {X -0.076,Y -161.203,Z 403.313,A 0.000,B 0.000,C 90.000,E1 236.421} C_DIS
LIN {X -0.040,Y -157.212,Z 403.289,A 0.000,B 0.000,C 90.000,E1 231.984} C_DIS
LIN {X -0.017,Y -155.939,Z 403.279,A 0.000,B 0.000,C 90.000,E1 230.194} C_DIS
LIN {X -0.057,Y -152.192,Z 403.254,A 0.000,B 0.000,C 90.000,E1 225.729} C_DIS
LIN {X -0.036,Y -150.438,Z 403.239,A 0.000,B 0.000,C 90.000,E1 223.014} C_DIS
LIN {X -0.009,Y -147.165,Z 403.214,A 0.000,B 0.000,C 90.000,E1 218.463} C_DIS
LIN {X -0.042,Y -145.180,Z 403.193,A 0.000,B 0.000,C 90.000,E1 214.818} C_DIS
LIN {X -0.007,Y -142.327,Z 403.163,A 0.000,B 0.000,C 90.000,E1 209.283} C_DIS
LIN {X -0.012,Y -141.716,Z 403.152,A 0.000,B 0.000,C 90.000,E1 207.436} C_DIS
LIN {X 0.036,Y -139.475,Z 403.116,A 0.000,B 0.000,C 90.000,E1 200.918} C_DIS
LIN {X 0.027,Y -138.970,Z 403.101,A 0.000,B 0.000,C 90.000,E1 198.127} C_DIS
LIN {X 0.016,Y -138.330,Z 403.054,A 0.000,B 0.000,C 90.000,E1 189.726} C_DIS
LIN {X 0.019,Y -139.436,Z 403.007,A 0.000,B 0.000,C 90.000,E1 181.318} C_DIS
LIN {X -0.041,Y -140.967,Z 402.976,A 0.000,B 0.000,C 90.000,E1 175.755} C_DIS
LIN {X 0.050,Y -142.722,Z 402.956,A 0.000,B 0.000,C 90.000,E1 172.008} C_DIS
LIN {X 0.007,Y -145.105,Z 402.930,A 0.000,B 0.000,C 90.000,E1 167.409} C_DIS
LIN {X 0.002,Y -147.729,Z 402.910,A 0.000,B 0.000,C 90.000,E1 163.740} C_DIS
LIN {X -0.057,Y -150.390,Z 402.889,A 0.000,B 0.000,C 90.000,E1 160.115} C_DIS
LIN {X -0.039,Y -153.823,Z 402.869,A 0.000,B 0.000,C 90.000,E1 156.485} C_DIS
LIN {X 0.019,Y -157.235,Z 402.849,A 0.000,B 0.000,C 90.000,E1 152.871} C_DIS
LIN {X -0.040,Y -161.404,Z 402.830,A 0.000,B 0.000,C 90.000,E1 149.331} C_DIS
LIN {X -0.031,Y -165.605,Z 402.810,A 0.000,B 0.000,C 90.000,E1 145.801} C_DIS
LIN {X 0.090,Y -170.531,Z 402.791,A 0.000,B 0.000,C 90.000,E1 142.271} C_DIS
LIN {X -0.001,Y -175.410,Z 402.771,A 0.000,B 0.000,C 90.000,E1 138.852} C_DIS
LIN {X -0.011,Y -181.034,Z 402.752,A 0.000,B 0.000,C 90.000,E1 135.445} C_DIS
LIN {X -0.017,Y -186.467,Z 402.734,A 0.000,B 0.000,C 90.000,E1 132.081} C_DIS
LIN {X 0.052,Y -191.090,Z 402.720,A 0.000,B 0.000,C 90.000,E1 129.564} C_DIS
LIN {X -0.025,Y -197.278,Z 402.700,A 0.000,B 0.000,C 90.000,E1 126.091} C_DIS
LIN {X -0.102,Y -197.477,Z 402.700,A 0.000,B 0.000,C 90.000,E1 126.011} C_DIS
LIN {X 0.039,Y -296.215,Z 402.700,A 0.000,B 0.000,C 90.000,E1 125.964} C_DIS
LIN {X -0.057,Y -297.705,Z 402.700,A 0.000,B 0.000,C 90.000,E1 125.964} C_DIS
LIN {X -0.058,Y -302.992,Z 402.698,A 0.000,B 0.000,C 90.000,E1 125.724} C_DIS
LIN {X 0.012,Y -305.689,Z 402.697,A 0.000,B 0.000,C 90.000,E1 125.471} C_DIS
LIN {X 0.071,Y -309.459,Z 402.694,A 0.000,B 0.000,C 90.000,E1 124.945} C_DIS
LIN {X 0.104,Y -311.137,Z 402.692,A 0.000,B 0.000,C 90.000,E1 124.612} C_DIS
LIN {X -0.121,Y -312.459,Z 402.691,A 0.000,B 0.000,C 90.000,E1 124.326} C_DIS
LIN {X 0.021,Y -323.538,Z 402.673,A 0.000,B 0.000,C 90.000,E1 121.082} C_DIS
LIN {X 0.079,Y -334.879,Z 402.657,A 0.000,B 0.000,C 90.000,E1 118.231} C_DIS
LIN {X -0.026,Y -347.656,Z 402.641,A 0.000,B 0.000,C 90.000,E1 115.463} C_DIS
LIN {X 0.055,Y -360.309,Z 402.628,A 0.000,B 0.000,C 90.000,E1 113.025} C_DIS
LIN {X -0.020,Y -374.278,Z 402.615,A 0.000,B 0.000,C 90.000,E1 110.663} C_DIS
LIN {X -0.152,Y -389.666,Z 402.602,A 0.000,B 0.000,C 90.000,E1 108.362} C_DIS
LIN {X -0.020,Y -406.586,Z 402.589,A 0.000,B 0.000,C 90.000,E1 106.079} C_DIS
LIN {X -0.088,Y -425.163,Z 402.577,A 0.000,B 0.000,C 90.000,E1 103.883} C_DIS
LIN {X -0.010,Y -445.120,Z 402.565,A 0.000,B 0.000,C 90.000,E1 101.771} C_DIS
LIN {X -0.056,Y -465.662,Z 402.555,A 0.000,B 0.000,C 90.000,E1 99.849} C_DIS
LIN {X 0.203,Y -486.702,Z 402.545,A 0.000,B 0.000,C 90.000,E1 98.049} C_DIS
LIN {X -0.063,Y -489.053,Z 402.544,A 0.000,B 0.000,C 90.000,E1 97.871} C_DIS
LIN {X 0.085,Y -490.836,Z 402.543,A 0.000,B 0.000,C 90.000,E1 97.644} C_DIS
LIN {X -0.017,Y -492.439,Z 402.541,A 0.000,B 0.000,C 90.000,E1 97.409} C_DIS
LIN {X -0.184,Y -493.640,Z 402.540,A 0.000,B 0.000,C 90.000,E1 97.182} C_DIS
LIN {X 0.055,Y -495.093,Z 402.537,A 0.000,B 0.000,C 90.000,E1 96.663} C_DIS
LIN {X -0.189,Y -495.493,Z 402.534,A 0.000,B 0.000,C 90.000,E1 96.201} C_DIS
LIN {X 0.065,Y -494.902,Z 402.532,A 0.000,B 0.000,C 90.000,E1 95.682} C_DIS
LIN {X -0.171,Y -493.223,Z 402.529,A 0.000,B 0.000,C 90.000,E1 95.220} C_DIS
LIN {X 0.179,Y -491.879,Z 402.528,A 0.000,B 0.000,C 90.000,E1 94.935} C_DIS
LIN {X -0.215,Y -486.400,Z 402.523,A 0.000,B 0.000,C 90.000,E1 94.245} C_DIS
LIN {X 0.000,Y -476.553,Z 402.517,A 0.000,B 0.000,C 90.000,E1 92.980} C_DIS
LIN {X -0.067,Y -457.108,Z 402.503,A 0.000,B 0.000,C 90.000,E1 90.458} C_DIS
LIN {X -0.025,Y -437.618,Z 402.487,A 0.000,B 0.000,C 90.000,E1 87.593} C_DIS
LIN {X 0.023,Y -418.115,Z 402.469,A 0.000,B 0.000,C 90.000,E1 84.375} C_DIS
LIN {X -0.055,Y -407.338,Z 402.458,A 0.000,B 0.000,C 90.000,E1 82.470} C_DIS
LIN {X -0.197,Y -393.698,Z 402.444,A 0.000,B 0.000,C 90.000,E1 79.982} C_DIS
LIN {X -0.148,Y -381.840,Z 402.432,A 0.000,B 0.000,C 90.000,E1 77.701} C_DIS
LIN {X 0.145,Y -368.802,Z 402.417,A 0.000,B 0.000,C 90.000,E1 75.046} C_DIS
LIN {X -0.072,Y -356.158,Z 402.402,A 0.000,B 0.000,C 90.000,E1 72.417} C_DIS
LIN {X -0.075,Y -344.091,Z 402.387,A 0.000,B 0.000,C 90.000,E1 69.699} C_DIS
LIN {X -0.039,Y -333.662,Z 402.373,A 0.000,B 0.000,C 90.000,E1 67.230} C_DIS
LIN {X 0.005,Y -323.581,Z 402.360,A 0.000,B 0.000,C 90.000,E1 64.717} C_DIS
LIN {X -0.001,Y -312.778,Z 402.344,A 0.000,B 0.000,C 90.000,E1 61.847} C_DIS
LIN {X 0.069,Y -300.257,Z 402.324,A 0.000,B 0.000,C 90.000,E1 58.250} C_DIS
LIN {X -0.015,Y -288.883,Z 402.303,A 0.000,B 0.000,C 90.000,E1 54.609} C_DIS
LIN {X -0.162,Y -279.403,Z 402.285,A 0.000,B 0.000,C 90.000,E1 51.251} C_DIS
LIN {X 0.086,Y -273.836,Z 402.273,A 0.000,B 0.000,C 90.000,E1 49.138} C_DIS
LIN {X 0.023,Y -268.099,Z 402.262,A 0.000,B 0.000,C 90.000,E1 47.067} C_DIS
LIN {X 0.028,Y -262.158,Z 402.250,A 0.000,B 0.000,C 90.000,E1 44.960} C_DIS
LIN {X -0.077,Y -256.144,Z 402.238,A 0.000,B 0.000,C 90.000,E1 42.852} C_DIS
LIN {X -0.097,Y -249.985,Z 402.226,A 0.000,B 0.000,C 90.000,E1 40.701} C_DIS
LIN {X 0.143,Y -241.827,Z 402.210,A 0.000,B 0.000,C 90.000,E1 37.729} C_DIS
LIN {X 0.048,Y -232.111,Z 402.189,A 0.000,B 0.000,C 90.000,E1 34.040} C_DIS
LIN {X 0.039,Y -223.324,Z 402.168,A 0.000,B 0.000,C 90.000,E1 30.256} C_DIS
LIN {X 0.007,Y -215.405,Z 402.147,A 0.000,B 0.000,C 90.000,E1 26.411} C_DIS
LIN {X -0.064,Y -208.595,Z 402.125,A 0.000,B 0.000,C 90.000,E1 22.514} C_DIS
LIN {X -0.071,Y -202.660,Z 402.103,A 0.000,B 0.000,C 90.000,E1 18.544} C_DIS
LIN {X 0.066,Y -197.740,Z 402.081,A 0.000,B 0.000,C 90.000,E1 14.481} C_DIS
LIN {X 0.007,Y -193.759,Z 402.058,A 0.000,B 0.000,C 90.000,E1 10.433} C_DIS
LIN {X 0.069,Y -190.939,Z 402.035,A 0.000,B 0.000,C 90.000,E1 6.315} C_DIS
LIN {X -0.034,Y -188.647,Z 401.997,A 0.000,B 0.000,C 90.000,E1 359.542} C_DIS
LIN {X -0.057,Y -190.464,Z 401.947,A 0.000,B 0.000,C 90.000,E1 350.443} C_DIS
LIN {X 0.073,Y -193.390,Z 401.919,A 0.000,B 0.000,C 90.000,E1 345.463} C_DIS
LIN {X -0.029,Y -196.895,Z 401.897,A 0.000,B 0.000,C 90.000,E1 341.402} C_DIS
LIN {X -0.076,Y -201.541,Z 401.874,A 0.000,B 0.000,C 90.000,E1 337.358} C_DIS
LIN {X -0.112,Y -206.008,Z 401.856,A 0.000,B 0.000,C 90.000,E1 334.152} C_DIS
LIN {X 0.074,Y -212.464,Z 401.834,A 0.000,B 0.000,C 90.000,E1 330.127} C_DIS
LIN {X 0.056,Y -219.558,Z 401.812,A 0.000,B 0.000,C 90.000,E1 326.215} C_DIS
LIN {X 0.079,Y -227.285,Z 401.791,A 0.000,B 0.000,C 90.000,E1 322.351} C_DIS
LIN {X 0.038,Y -235.941,Z 401.770,A 0.000,B 0.000,C 90.000,E1 318.566} C_DIS
LIN {X -0.102,Y -244.789,Z 401.751,A 0.000,B 0.000,C 90.000,E1 315.243} C_DIS
LIN {X 0.046,Y -254.887,Z 401.733,A 0.000,B 0.000,C 90.000,E1 311.919} C_DIS
LIN {X 0.014,Y -266.315,Z 401.715,A 0.000,B 0.000,C 90.000,E1 308.705} C_DIS
LIN {X -0.038,Y -278.422,Z 401.698,A 0.000,B 0.000,C 90.000,E1 305.564} C_DIS
LIN {X -0.075,Y -289.810,Z 401.682,A 0.000,B 0.000,C 90.000,E1 302.832} C_DIS
LIN {X 0.067,Y -304.954,Z 401.664,A 0.000,B 0.000,C 90.000,E1 299.461} C_DIS
LIN {X 0.048,Y -316.799,Z 401.651,A 0.000,B 0.000,C 90.000,E1 297.180} C_DIS
LIN {X -0.003,Y -329.649,Z 401.639,A 0.000,B 0.000,C 90.000,E1 294.951} C_DIS
LIN {X -0.037,Y -345.940,Z 401.625,A 0.000,B 0.000,C 90.000,E1 292.461} C_DIS
LIN {X 0.226,Y -363.666,Z 401.611,A 0.000,B 0.000,C 90.000,E1 289.993} C_DIS
LIN {X 0.116,Y -380.134,Z 401.600,A 0.000,B 0.000,C 90.000,E1 287.946} C_DIS
LIN {X -0.189,Y -405.755,Z 401.584,A 0.000,B 0.000,C 90.000,E1 285.190} C_DIS
LIN {X 0.042,Y -421.481,Z 401.576,A 0.000,B 0.000,C 90.000,E1 283.592} C_DIS
LIN {X 0.113,Y -434.336,Z 401.568,A 0.000,B 0.000,C 90.000,E1 282.299} C_DIS
LIN {X 0.201,Y -441.602,Z 401.564,A 0.000,B 0.000,C 90.000,E1 281.535} C_DIS
LIN {X 0.083,Y -448.466,Z 401.560,A 0.000,B 0.000,C 90.000,E1 280.782} C_DIS
LIN {X -0.075,Y -454.932,Z 401.556,A 0.000,B 0.000,C 90.000,E1 280.018} C_DIS
LIN {X 0.013,Y -462.720,Z 401.550,A 0.000,B 0.000,C 90.000,E1 278.973} C_DIS
LIN {X 0.128,Y -469.792,Z 401.544,A 0.000,B 0.000,C 90.000,E1 277.936} C_DIS
LIN {X -0.077,Y -476.240,Z 401.539,A 0.000,B 0.000,C 90.000,E1 276.947} C_DIS
LIN {X -0.142,Y -480.588,Z 401.534,A 0.000,B 0.000,C 90.000,E1 276.201} C_DIS
LIN {X -0.114,Y -484.345,Z 401.530,A 0.000,B 0.000,C 90.000,E1 275.448} C_DIS
LIN {X 0.191,Y -485.457,Z 401.529,A 0.000,B 0.000,C 90.000,E1 275.163} C_DIS
LIN {X -0.105,Y -487.349,Z 401.526,A 0.000,B 0.000,C 90.000,E1 274.702} C_DIS
LIN {X 0.050,Y -488.828,Z 401.523,A 0.000,B 0.000,C 90.000,E1 274.188} C_DIS
LIN {X -0.233,Y -489.978,Z 401.521,A 0.000,B 0.000,C 90.000,E1 273.726} C_DIS
LIN {X -0.051,Y -490.814,Z 401.518,A 0.000,B 0.000,C 90.000,E1 273.212} C_DIS
LIN {X 0.165,Y -491.362,Z 401.515,A 0.000,B 0.000,C 90.000,E1 272.694} C_DIS
LIN {X -0.129,Y -491.571,Z 401.512,A 0.000,B 0.000,C 90.000,E1 272.236} C_DIS
LIN {X 0.090,Y -491.459,Z 401.510,A 0.000,B 0.000,C 90.000,E1 271.718} C_DIS
LIN {X -0.199,Y -490.970,Z 401.507,A 0.000,B 0.000,C 90.000,E1 271.260} C_DIS
LIN {X 0.005,Y -490.058,Z 401.504,A 0.000,B 0.000,C 90.000,E1 270.745} C_DIS
LIN {X 0.206,Y -488.629,Z 401.501,A 0.000,B 0.000,C 90.000,E1 270.229} C_DIS
LIN {X -0.087,Y -486.710,Z 401.499,A 0.000,B 0.000,C 90.000,E1 269.771} C_DIS
LIN {X 0.099,Y -484.119,Z 401.496,A 0.000,B 0.000,C 90.000,E1 269.255} C_DIS
LIN {X -0.217,Y -480.735,Z 401.493,A 0.000,B 0.000,C 90.000,E1 268.797} C_DIS
LIN {X 0.097,Y -478.702,Z 401.492,A 0.000,B 0.000,C 90.000,E1 268.511} C_DIS
LIN {X -0.227,Y -473.793,Z 401.489,A 0.000,B 0.000,C 90.000,E1 268.051} C_DIS
LIN {X 0.072,Y -470.896,Z 401.488,A 0.000,B 0.000,C 90.000,E1 267.764} C_DIS
LIN {X 0.104,Y -467.873,Z 401.486,A 0.000,B 0.000,C 90.000,E1 267.535} C_DIS
LIN {X 0.030,Y -461.232,Z 401.484,A 0.000,B 0.000,C 90.000,E1 267.135} C_DIS
LIN {X 0.151,Y -454.239,Z 401.482,A 0.000,B 0.000,C 90.000,E1 266.788} C_DIS
LIN {X -0.170,Y -447.139,Z 401.481,A 0.000,B 0.000,C 90.000,E1 266.560} C_DIS
LIN {X -0.111,Y -439.777,Z 401.480,A 0.000,B 0.000,C 90.000,E1 266.331} C_DIS
LIN {X -0.135,Y -431.724,Z 401.479,A 0.000,B 0.000,C 90.000,E1 266.159} C_DIS
LIN {X 0.180,Y -422.285,Z 401.478,A 0.000,B 0.000,C 90.000,E1 265.988} C_DIS
LIN {X 0.113,Y -411.600,Z 401.477,A 0.000,B 0.000,C 90.000,E1 265.927} C_DIS
LIN {X 0.022,Y -180.917,Z 401.477,A 0.000,B 0.000,C 90.000,E1 265.927} C_DIS
LIN {X -0.056,Y -180.872,Z 401.472,A 0.000,B 0.000,C 90.000,E1 265.065} C_DIS
LIN {X 0.001,Y -178.988,Z 401.444,A 0.000,B 0.000,C 90.000,E1 259.982} C_DIS
LIN {X 0.013,Y -177.970,Z 401.435,A 0.000,B 0.000,C 90.000,E1 258.285} C_DIS
LIN {X 0.031,Y -175.613,Z 401.411,A 0.000,B 0.000,C 90.000,E1 254.031} C_DIS
LIN {X 0.044,Y -172.335,Z 401.388,A 0.000,B 0.000,C 90.000,E1 249.752} C_DIS
LIN {X 0.022,Y -171.812,Z 401.383,A 0.000,B 0.000,C 90.000,E1 248.901} C_DIS
LIN {X 0.029,Y -170.275,Z 401.373,A 0.000,B 0.000,C 90.000,E1 247.177} C_DIS
LIN {X -0.034,Y -166.816,Z 401.349,A 0.000,B 0.000,C 90.000,E1 242.871} C_DIS
LIN {X 0.023,Y -162.799,Z 401.325,A 0.000,B 0.000,C 90.000,E1 238.486} C_DIS
LIN {X -0.052,Y -161.485,Z 401.315,A 0.000,B 0.000,C 90.000,E1 236.755} C_DIS
LIN {X -0.001,Y -157.481,Z 401.291,A 0.000,B 0.000,C 90.000,E1 232.316} C_DIS
LIN {X 0.055,Y -155.498,Z 401.276,A 0.000,B 0.000,C 90.000,E1 229.622} C_DIS
LIN {X -0.012,Y -151.802,Z 401.251,A 0.000,B 0.000,C 90.000,E1 225.162} C_DIS
LIN {X 0.000,Y -150.014,Z 401.236,A 0.000,B 0.000,C 90.000,E1 222.447} C_DIS
LIN {X 0.031,Y -146.838,Z 401.211,A 0.000,B 0.000,C 90.000,E1 217.890} C_DIS
LIN {X 0.018,Y -145.419,Z 401.195,A 0.000,B 0.000,C 90.000,E1 215.152} C_DIS
LIN {X 0.053,Y -142.847,Z 401.170,A 0.000,B 0.000,C 90.000,E1 210.541} C_DIS
LIN {X -0.017,Y -141.461,Z 401.149,A 0.000,B 0.000,C 90.000,E1 206.873} C_DIS
LIN {X -0.027,Y -139.375,Z 401.113,A 0.000,B 0.000,C 90.000,E1 200.375} C_DIS
LIN {X -0.036,Y -138.826,Z 401.098,A 0.000,B 0.000,C 90.000,E1 197.583} C_DIS
LIN {X 0.053,Y -138.353,Z 401.056,A 0.000,B 0.000,C 90.000,E1 190.074} C_DIS
LIN {X 0.026,Y -139.530,Z 401.004,A 0.000,B 0.000,C 90.000,E1 180.745} C_DIS
LIN {X -0.021,Y -141.208,Z 400.973,A 0.000,B 0.000,C 90.000,E1 175.179} C_DIS
LIN {X -0.062,Y -142.583,Z 400.958,A 0.000,B 0.000,C 90.000,E1 172.413} C_DIS
LIN {X 0.033,Y -144.879,Z 400.932,A 0.000,B 0.000,C 90.000,E1 167.757} C_DIS
LIN {X -0.012,Y -147.506,Z 400.912,A 0.000,B 0.000,C 90.000,E1 164.102} C_DIS
LIN {X 0.062,Y -150.099,Z 400.891,A 0.000,B 0.000,C 90.000,E1 160.423} C_DIS
LIN {X 0.075,Y -153.454,Z 400.871,A 0.000,B 0.000,C 90.000,E1 156.794} C_DIS
LIN {X -0.074,Y -157.818,Z 400.846,A 0.000,B 0.000,C 90.000,E1 152.359} C_DIS
LIN {X -0.042,Y -162.100,Z 400.827,A 0.000,B 0.000,C 90.000,E1 148.791} C_DIS
LIN {X -0.018,Y -166.300,Z 400.807,A 0.000,B 0.000,C 90.000,E1 145.261} C_DIS
LIN {X -0.020,Y -171.318,Z 400.788,A 0.000,B 0.000,C 90.000,E1 141.778} C_DIS
LIN {X 0.014,Y -176.217,Z 400.768,A 0.000,B 0.000,C 90.000,E1 138.324} C_DIS
LIN {X 0.008,Y -180.494,Z 400.754,A 0.000,B 0.000,C 90.000,E1 135.769} C_DIS
LIN {X -0.011,Y -185.898,Z 400.736,A 0.000,B 0.000,C 90.000,E1 132.405} C_DIS
LIN {X 0.050,Y -190.525,Z 400.722,A 0.000,B 0.000,C 90.000,E1 129.886} C_DIS
LIN {X -0.012,Y -197.582,Z 400.700,A 0.000,B 0.000,C 90.000,E1 125.931} C_DIS
LIN {X -0.052,Y -296.367,Z 400.700,A 0.000,B 0.000,C 90.000,E1 125.931} C_DIS
LIN {X 0.118,Y -297.595,Z 400.699,A 0.000,B 0.000,C 90.000,E1 125.884} C_DIS
LIN {X -0.072,Y -301.054,Z 400.699,A 0.000,B 0.000,C 90.000,E1 125.804} C_DIS
LIN {X -0.103,Y -304.195,Z 400.698,A 0.000,B 0.000,C 90.000,E1 125.598} C_DIS
LIN {X -0.069,Y -307.893,Z 400.695,A 0.000,B 0.000,C 90.000,E1 125.185} C_DIS
LIN {X -0.162,Y -309.825,Z 400.694,A 0.000,B 0.000,C 90.000,E1 124.898} C_DIS
LIN {X 0.001,Y -311.349,Z 400.692,A 0.000,B 0.000,C 90.000,E1 124.565} C_DIS
LIN {X 0.011,Y -313.711,Z 400.688,A 0.000,B 0.000,C 90.000,E1 123.913} C_DIS
LIN {X 0.112,Y -323.750,Z 400.672,A 0.000,B 0.000,C 90.000,E1 121.003} C_DIS
LIN {X 0.010,Y -335.124,Z 400.657,A 0.000,B 0.000,C 90.000,E1 118.180} C_DIS
LIN {X -0.079,Y -347.930,Z 400.641,A 0.000,B 0.000,C 90.000,E1 115.412} C_DIS
LIN {X 0.155,Y -360.614,Z 400.628,A 0.000,B 0.000,C 90.000,E1 112.950} C_DIS
LIN {X -0.049,Y -374.617,Z 400.614,A 0.000,B 0.000,C 90.000,E1 110.610} C_DIS
LIN {X -0.046,Y -390.040,Z 400.602,A 0.000,B 0.000,C 90.000,E1 108.290} C_DIS
LIN {X -0.022,Y -406.999,Z 400.589,A 0.000,B 0.000,C 90.000,E1 106.024} C_DIS
LIN {X -0.075,Y -425.618,Z 400.577,A 0.000,B 0.000,C 90.000,E1 103.828} C_DIS
LIN {X 0.047,Y -445.582,Z 400.565,A 0.000,B 0.000,C 90.000,E1 101.715} C_DIS
LIN {X 0.038,Y -466.138,Z 400.554,A 0.000,B 0.000,C 90.000,E1 99.792} C_DIS
LIN {X -0.147,Y -487.189,Z 400.545,A 0.000,B 0.000,C 90.000,E1 98.049} C_DIS
LIN {X 0.053,Y -489.483,Z 400.543,A 0.000,B 0.000,C 90.000,E1 97.814} C_DIS
LIN {X 0.013,Y -491.371,Z 400.542,A 0.000,B 0.000,C 90.000,E1 97.587} C_DIS
LIN {X 0.038,Y -492.808,Z 400.541,A 0.000,B 0.000,C 90.000,E1 97.352} C_DIS
LIN {X -0.221,Y -494.788,Z 400.538,A 0.000,B 0.000,C 90.000,E1 96.891} C_DIS
LIN {X 0.019,Y -495.626,Z 400.535,A 0.000,B 0.000,C 90.000,E1 96.372} C_DIS
LIN {X -0.221,Y -495.463,Z 400.533,A 0.000,B 0.000,C 90.000,E1 95.910} C_DIS
LIN {X 0.035,Y -494.277,Z 400.530,A 0.000,B 0.000,C 90.000,E1 95.391} C_DIS
LIN {X -0.107,Y -493.242,Z 400.529,A 0.000,B 0.000,C 90.000,E1 95.163} C_DIS
LIN {X -0.246,Y -491.842,Z 400.527,A 0.000,B 0.000,C 90.000,E1 94.935} C_DIS
LIN {X 0.213,Y -484.409,Z 400.522,A 0.000,B 0.000,C 90.000,E1 93.898} C_DIS
LIN {X 0.184,Y -472.484,Z 400.513,A 0.000,B 0.000,C 90.000,E1 92.407} C_DIS
LIN {X 0.005,Y -453.378,Z 400.499,A 0.000,B 0.000,C 90.000,E1 89.885} C_DIS
LIN {X -0.079,Y -434.189,Z 400.483,A 0.000,B 0.000,C 90.000,E1 87.020} C_DIS
LIN {X -0.117,Y -414.969,Z 400.465,A 0.000,B 0.000,C 90.000,E1 83.799} C_DIS
LIN {X 0.149,Y -404.237,Z 400.455,A 0.000,B 0.000,C 90.000,E1 81.837} C_DIS
LIN {X -0.029,Y -390.677,Z 400.441,A 0.000,B 0.000,C 90.000,E1 79.342} C_DIS
LIN {X -0.084,Y -380.332,Z 400.430,A 0.000,B 0.000,C 90.000,E1 77.353} C_DIS
LIN {X 0.175,Y -368.801,Z 400.417,A 0.000,B 0.000,C 90.000,E1 74.991} C_DIS
LIN {X -0.053,Y -356.122,Z 400.402,A 0.000,B 0.000,C 90.000,E1 72.362} C_DIS
LIN {X 0.060,Y -344.020,Z 400.387,A 0.000,B 0.000,C 90.000,E1 69.625} C_DIS
LIN {X -0.048,Y -332.250,Z 400.371,A 0.000,B 0.000,C 90.000,E1 66.869} C_DIS
LIN {X -0.016,Y -319.789,Z 400.354,A 0.000,B 0.000,C 90.000,E1 63.717} C_DIS
LIN {X -0.114,Y -309.116,Z 400.338,A 0.000,B 0.000,C 90.000,E1 60.845} C_DIS
LIN {X 0.083,Y -297.971,Z 400.320,A 0.000,B 0.000,C 90.000,E1 57.533} C_DIS
LIN {X 0.100,Y -287.793,Z 400.301,A 0.000,B 0.000,C 90.000,E1 54.196} C_DIS
LIN {X 0.083,Y -278.351,Z 400.282,A 0.000,B 0.000,C 90.000,E1 50.803} C_DIS
LIN {X -0.079,Y -272.785,Z 400.271,A 0.000,B 0.000,C 90.000,E1 48.771} C_DIS
LIN {X 0.022,Y -267.018,Z 400.259,A 0.000,B 0.000,C 90.000,E1 46.662} C_DIS
LIN {X 0.005,Y -261.098,Z 400.248,A 0.000,B 0.000,C 90.000,E1 44.555} C_DIS
LIN {X -0.118,Y -255.076,Z 400.236,A 0.000,B 0.000,C 90.000,E1 42.447} C_DIS
LIN {X 0.030,Y -248.930,Z 400.224,A 0.000,B 0.000,C 90.000,E1 40.253} C_DIS
LIN {X -0.101,Y -240.811,Z 400.207,A 0.000,B 0.000,C 90.000,E1 37.363} C_DIS
LIN {X -0.030,Y -231.190,Z 400.187,A 0.000,B 0.000,C 90.000,E1 33.627} C_DIS
LIN {X 0.127,Y -222.479,Z 400.166,A 0.000,B 0.000,C 90.000,E1 29.795} C_DIS
LIN {X -0.032,Y -214.639,Z 400.144,A 0.000,B 0.000,C 90.000,E1 25.976} C_DIS
LIN {X 0.071,Y -207.901,Z 400.122,A 0.000,B 0.000,C 90.000,E1 22.025} C_DIS
LIN {X 0.039,Y -202.066,Z 400.100,A 0.000,B 0.000,C 90.000,E1 18.055} C_DIS
LIN {X -0.092,Y -197.234,Z 400.078,A 0.000,B 0.000,C 90.000,E1 14.064} C_DIS
LIN {X 0.020,Y -193.301,Z 400.055,A 0.000,B 0.000,C 90.000,E1 9.962} C_DIS
LIN {X -0.029,Y -190.190,Z 400.028,A 0.000,B 0.000,C 90.000,E1 5.049} C_DIS
LIN {X -0.014,Y -188.492,Z 399.988,A 0.000,B 0.000,C 90.000,E1 357.879} C_DIS
LIN {X -0.063,Y -190.349,Z 399.947,A 0.000,B 0.000,C 90.000,E1 350.443} C_DIS
LIN {X 0.061,Y -193.269,Z 399.919,A 0.000,B 0.000,C 90.000,E1 345.463} C_DIS
LIN {X -0.043,Y -196.761,Z 399.897,A 0.000,B 0.000,C 90.000,E1 341.402} C_DIS
LIN {X -0.096,Y -201.399,Z 399.874,A 0.000,B 0.000,C 90.000,E1 337.358} C_DIS
LIN {X 0.049,Y -205.878,Z 399.856,A 0.000,B 0.000,C 90.000,E1 334.101} C_DIS
LIN {X 0.046,Y -212.353,Z 399.834,A 0.000,B 0.000,C 90.000,E1 330.127} C_DIS
LIN {X 0.023,Y -219.431,Z 399.812,A 0.000,B 0.000,C 90.000,E1 326.215} C_DIS
LIN {X 0.040,Y -227.167,Z 399.791,A 0.000,B 0.000,C 90.000,E1 322.351} C_DIS
LIN {X -0.005,Y -235.832,Z 399.770,A 0.000,B 0.000,C 90.000,E1 318.566} C_DIS
LIN {X 0.030,Y -244.691,Z 399.751,A 0.000,B 0.000,C 90.000,E1 315.202} C_DIS
LIN {X -0.002,Y -254.793,Z 399.733,A 0.000,B 0.000,C 90.000,E1 311.919} C_DIS
LIN {X -0.038,Y -266.249,Z 399.715,A 0.000,B 0.000,C 90.000,E1 308.705} C_DIS
LIN {X 0.132,Y -278.320,Z 399.697,A 0.000,B 0.000,C 90.000,E1 305.518} C_DIS
LIN {X -0.106,Y -288.258,Z 399.684,A 0.000,B 0.000,C 90.000,E1 303.166} C_DIS
LIN {X -0.017,Y -303.290,Z 399.665,A 0.000,B 0.000,C 90.000,E1 299.795} C_DIS
LIN {X -0.079,Y -315.007,Z 399.653,A 0.000,B 0.000,C 90.000,E1 297.513} C_DIS
LIN {X -0.078,Y -329.669,Z 399.639,A 0.000,B 0.000,C 90.000,E1 294.951} C_DIS
LIN {X -0.114,Y -346.067,Z 399.625,A 0.000,B 0.000,C 90.000,E1 292.461} C_DIS
LIN {X 0.148,Y -363.804,Z 399.611,A 0.000,B 0.000,C 90.000,E1 289.993} C_DIS
LIN {X 0.039,Y -380.350,Z 399.600,A 0.000,B 0.000,C 90.000,E1 287.946} C_DIS
LIN {X 0.061,Y -403.275,Z 399.586,A 0.000,B 0.000,C 90.000,E1 285.426} C_DIS
LIN {X 0.166,Y -421.458,Z 399.576,A 0.000,B 0.000,C 90.000,E1 283.592} C_DIS
LIN {X 0.217,Y -434.288,Z 399.568,A 0.000,B 0.000,C 90.000,E1 282.299} C_DIS
LIN {X 0.149,Y -441.708,Z 399.564,A 0.000,B 0.000,C 90.000,E1 281.535} C_DIS
LIN {X -0.117,Y -448.717,Z 399.560,A 0.000,B 0.000,C 90.000,E1 280.782} C_DIS
LIN {X 0.173,Y -455.161,Z 399.555,A 0.000,B 0.000,C 90.000,E1 279.962} C_DIS
LIN {X -0.012,Y -461.030,Z 399.551,A 0.000,B 0.000,C 90.000,E1 279.208} C_DIS
LIN {X -0.144,Y -466.515,Z 399.547,A 0.000,B 0.000,C 90.000,E1 278.454} C_DIS
LIN {X 0.080,Y -473.231,Z 399.541,A 0.000,B 0.000,C 90.000,E1 277.409} C_DIS
LIN {X -0.011,Y -477.880,Z 399.537,A 0.000,B 0.000,C 90.000,E1 276.663} C_DIS
LIN {X -0.003,Y -482.024,Z 399.533,A 0.000,B 0.000,C 90.000,E1 275.910} C_DIS
LIN {X -0.013,Y -485.530,Z 399.529,A 0.000,B 0.000,C 90.000,E1 275.163} C_DIS
LIN {X 0.176,Y -487.399,Z 399.526,A 0.000,B 0.000,C 90.000,E1 274.645} C_DIS
LIN {X -0.155,Y -488.845,Z 399.523,A 0.000,B 0.000,C 90.000,E1 274.188} C_DIS
LIN {X 0.050,Y -489.982,Z 399.520,A 0.000,B 0.000,C 90.000,E1 273.669} C_DIS
LIN {X -0.258,Y -490.826,Z 399.518,A 0.000,B 0.000,C 90.000,E1 273.212} C_DIS
LIN {X -0.041,Y -491.341,Z 399.515,A 0.000,B 0.000,C 90.000,E1 272.694} C_DIS
LIN {X 0.157,Y -491.505,Z 399.512,A 0.000,B 0.000,C 90.000,E1 272.178} C_DIS
LIN {X -0.116,Y -491.395,Z 399.509,A 0.000,B 0.000,C 90.000,E1 271.718} C_DIS
LIN {X 0.086,Y -490.881,Z 399.507,A 0.000,B 0.000,C 90.000,E1 271.203} C_DIS
LIN {X -0.201,Y -489.920,Z 399.504,A 0.000,B 0.000,C 90.000,E1 270.745} C_DIS
LIN {X 0.000,Y -488.540,Z 399.501,A 0.000,B 0.000,C 90.000,E1 270.229} C_DIS
LIN {X 0.194,Y -486.612,Z 399.499,A 0.000,B 0.000,C 90.000,E1 269.714} C_DIS
LIN {X -0.106,Y -483.975,Z 399.496,A 0.000,B 0.000,C 90.000,E1 269.255} C_DIS
LIN {X 0.059,Y -480.572,Z 399.493,A 0.000,B 0.000,C 90.000,E1 268.740} C_DIS
LIN {X 0.204,Y -476.198,Z 399.490,A 0.000,B 0.000,C 90.000,E1 268.224} C_DIS
LIN {X 0.044,Y -473.579,Z 399.489,A 0.000,B 0.000,C 90.000,E1 267.993} C_DIS
LIN {X -0.131,Y -470.616,Z 399.487,A 0.000,B 0.000,C 90.000,E1 267.764} C_DIS
LIN {X -0.071,Y -467.624,Z 399.486,A 0.000,B 0.000,C 90.000,E1 267.535} C_DIS
LIN {X -0.099,Y -460.965,Z 399.484,A 0.000,B 0.000,C 90.000,E1 267.135} C_DIS
LIN {X 0.039,Y -454.014,Z 399.482,A 0.000,B 0.000,C 90.000,E1 266.788} C_DIS
LIN {X 0.175,Y -446.890,Z 399.481,A 0.000,B 0.000,C 90.000,E1 266.502} C_DIS
LIN {X -0.204,Y -439.501,Z 399.479,A 0.000,B 0.000,C 90.000,E1 266.331} C_DIS
LIN {X -0.203,Y -431.412,Z 399.479,A 0.000,B 0.000,C 90.000,E1 266.159} C_DIS
LIN {X 0.146,Y -422.281,Z 399.478,A 0.000,B 0.000,C 90.000,E1 265.988} C_DIS
LIN {X 0.182,Y -415.533,Z 399.478,A 0.000,B 0.000,C 90.000,E1 265.931} C_DIS
LIN {X 0.094,Y -411.542,Z 399.477,A 0.000,B 0.000,C 90.000,E1 265.927} C_DIS
LIN {X 0.015,Y -180.917,Z 399.477,A 0.000,B 0.000,C 90.000,E1 265.927} C_DIS
LIN {X -0.053,Y -180.872,Z 399.473,A 0.000,B 0.000,C 90.000,E1 265.065} C_DIS
LIN {X 0.003,Y -178.988,Z 399.444,A 0.000,B 0.000,C 90.000,E1 259.982} C_DIS
LIN {X 0.015,Y -177.971,Z 399.435,A 0.000,B 0.000,C 90.000,E1 258.285} C_DIS
LIN {X 0.034,Y -175.614,Z 399.411,A 0.000,B 0.000,C 90.000,E1 254.031} C_DIS
LIN {X 0.046,Y -172.335,Z 399.388,A 0.000,B 0.000,C 90.000,E1 249.752} C_DIS
LIN {X 0.024,Y -171.812,Z 399.383,A 0.000,B 0.000,C 90.000,E1 248.901} C_DIS
LIN {X 0.032,Y -170.275,Z 399.373,A 0.000,B 0.000,C 90.000,E1 247.177} C_DIS
LIN {X -0.032,Y -166.817,Z 399.349,A 0.000,B 0.000,C 90.000,E1 242.871} C_DIS
LIN {X 0.025,Y -162.798,Z 399.325,A 0.000,B 0.000,C 90.000,E1 238.486} C_DIS
LIN {X -0.049,Y -161.486,Z 399.315,A 0.000,B 0.000,C 90.000,E1 236.755} C_DIS
LIN {X 0.001,Y -157.482,Z 399.291,A 0.000,B 0.000,C 90.000,E1 232.316} C_DIS
LIN {X 0.057,Y -155.499,Z 399.276,A 0.000,B 0.000,C 90.000,E1 229.622} C_DIS
LIN {X -0.010,Y -151.803,Z 399.251,A 0.000,B 0.000,C 90.000,E1 225.162} C_DIS
LIN {X 0.002,Y -150.014,Z 399.236,A 0.000,B 0.000,C 90.000,E1 222.447} C_DIS
LIN {X 0.033,Y -146.838,Z 399.211,A 0.000,B 0.000,C 90.000,E1 217.890} C_DIS
LIN {X 0.019,Y -145.420,Z 399.195,A 0.000,B 0.000,C 90.000,E1 215.152} C_DIS
LIN {X 0.055,Y -142.847,Z 399.170,A 0.000,B 0.000,C 90.000,E1 210.541} C_DIS
LIN {X -0.015,Y -141.461,Z 399.149,A 0.000,B 0.000,C 90.000,E1 206.873} C_DIS
LIN {X -0.025,Y -139.375,Z 399.113,A 0.000,B 0.000,C 90.000,E1 200.375} C_DIS
LIN {X -0.034,Y -138.826,Z 399.098,A 0.000,B 0.000,C 90.000,E1 197.583} C_DIS
LIN {X 0.054,Y -138.353,Z 399.056,A 0.000,B 0.000,C 90.000,E1 190.074} C_DIS
LIN {X 0.028,Y -139.530,Z 399.004,A 0.000,B 0.000,C 90.000,E1 180.745} C_DIS
LIN {X -0.019,Y -141.208,Z 398.973,A 0.000,B 0.000,C 90.000,E1 175.179} C_DIS
LIN {X -0.060,Y -142.583,Z 398.958,A 0.000,B 0.000,C 90.000,E1 172.413} C_DIS
LIN {X 0.035,Y -144.878,Z 398.932,A 0.000,B 0.000,C 90.000,E1 167.757} C_DIS
LIN {X -0.010,Y -147.506,Z 398.912,A 0.000,B 0.000,C 90.000,E1 164.102} C_DIS
LIN {X 0.064,Y -150.098,Z 398.891,A 0.000,B 0.000,C 90.000,E1 160.423} C_DIS
LIN {X 0.077,Y -153.453,Z 398.871,A 0.000,B 0.000,C 90.000,E1 156.794} C_DIS
LIN {X -0.071,Y -157.816,Z 398.846,A 0.000,B 0.000,C 90.000,E1 152.359} C_DIS
LIN {X -0.039,Y -162.099,Z 398.827,A 0.000,B 0.000,C 90.000,E1 148.791} C_DIS
LIN {X -0.015,Y -166.299,Z 398.807,A 0.000,B 0.000,C 90.000,E1 145.261} C_DIS
LIN {X -0.019,Y -171.317,Z 398.788,A 0.000,B 0.000,C 90.000,E1 141.778} C_DIS
LIN {X 0.016,Y -176.216,Z 398.768,A 0.000,B 0.000,C 90.000,E1 138.324} C_DIS
LIN {X 0.010,Y -180.493,Z 398.754,A 0.000,B 0.000,C 90.000,E1 135.769} C_DIS
LIN {X -0.008,Y -185.896,Z 398.736,A 0.000,B 0.000,C 90.000,E1 132.405} C_DIS
LIN {X 0.053,Y -190.524,Z 398.722,A 0.000,B 0.000,C 90.000,E1 129.886} C_DIS
LIN {X 0.068,Y -197.627,Z 398.699,A 0.000,B 0.000,C 90.000,E1 125.884} C_DIS
LIN {X -0.025,Y -197.680,Z 398.699,A 0.000,B 0.000,C 90.000,E1 125.884} C_DIS
LIN {X -0.073,Y -296.415,Z 398.699,A 0.000,B 0.000,C 90.000,E1 125.884} C_DIS
LIN {X -0.005,Y -298.080,Z 398.699,A 0.000,B 0.000,C 90.000,E1 125.851} C_DIS
LIN {X -0.068,Y -300.050,Z 398.699,A 0.000,B 0.000,C 90.000,E1 125.804} C_DIS
LIN {X 0.024,Y -303.399,Z 398.698,A 0.000,B 0.000,C 90.000,E1 125.598} C_DIS
LIN {X 0.134,Y -306.986,Z 398.696,A 0.000,B 0.000,C 90.000,E1 125.231} C_DIS
LIN {X 0.087,Y -310.558,Z 398.693,A 0.000,B 0.000,C 90.000,E1 124.692} C_DIS
LIN {X -0.133,Y -312.059,Z 398.691,A 0.000,B 0.000,C 90.000,E1 124.405} C_DIS
LIN {X 0.120,Y -318.627,Z 398.680,A 0.000,B 0.000,C 90.000,E1 122.418} C_DIS
LIN {X -0.089,Y -329.332,Z 398.664,A 0.000,B 0.000,C 90.000,E1 119.589} C_DIS
LIN {X 0.101,Y -341.418,Z 398.649,A 0.000,B 0.000,C 90.000,E1 116.744} C_DIS
LIN {X -0.151,Y -353.413,Z 398.635,A 0.000,B 0.000,C 90.000,E1 114.335} C_DIS
LIN {X 0.077,Y -366.673,Z 398.622,A 0.000,B 0.000,C 90.000,E1 111.897} C_DIS
LIN {X -0.111,Y -381.296,Z 398.609,A 0.000,B 0.000,C 90.000,E1 109.577} C_DIS
LIN {X -0.065,Y -397.391,Z 398.596,A 0.000,B 0.000,C 90.000,E1 107.275} C_DIS
LIN {X 0.150,Y -415.073,Z 398.583,A 0.000,B 0.000,C 90.000,E1 105.009} C_DIS
LIN {X -0.181,Y -434.422,Z 398.571,A 0.000,B 0.000,C 90.000,E1 102.883} C_DIS
LIN {X 0.018,Y -454.673,Z 398.560,A 0.000,B 0.000,C 90.000,E1 100.838} C_DIS
LIN {X 0.138,Y -475.459,Z 398.550,A 0.000,B 0.000,C 90.000,E1 98.973} C_DIS
LIN {X -0.224,Y -488.604,Z 398.544,A 0.000,B 0.000,C 90.000,E1 97.936} C_DIS
LIN {X 0.031,Y -492.186,Z 398.542,A 0.000,B 0.000,C 90.000,E1 97.473} C_DIS
LIN {X -0.073,Y -493.544,Z 398.540,A 0.000,B 0.000,C 90.000,E1 97.239} C_DIS
LIN {X -0.180,Y -494.548,Z 398.539,A 0.000,B 0.000,C 90.000,E1 97.004} C_DIS
LIN {X 0.064,Y -495.673,Z 398.536,A 0.000,B 0.000,C 90.000,E1 96.486} C_DIS
LIN {X -0.180,Y -495.782,Z 398.533,A 0.000,B 0.000,C 90.000,E1 96.024} C_DIS
LIN {X 0.029,Y -494.891,Z 398.531,A 0.000,B 0.000,C 90.000,E1 95.511} C_DIS
LIN {X -0.205,Y -492.842,Z 398.528,A 0.000,B 0.000,C 90.000,E1 95.049} C_DIS
LIN {X 0.045,Y -489.453,Z 398.525,A 0.000,B 0.000,C 90.000,E1 94.531} C_DIS
LIN {X -0.044,Y -481.791,Z 398.520,A 0.000,B 0.000,C 90.000,E1 93.555} C_DIS
LIN {X 0.053,Y -462.076,Z 398.506,A 0.000,B 0.000,C 90.000,E1 91.031} C_DIS
LIN {X -0.220,Y -442.078,Z 398.490,A 0.000,B 0.000,C 90.000,E1 88.224} C_DIS
LIN {X -0.023,Y -422.202,Z 398.472,A 0.000,B 0.000,C 90.000,E1 85.008} C_DIS
LIN {X 0.058,Y -409.849,Z 398.460,A 0.000,B 0.000,C 90.000,E1 82.818} C_DIS
LIN {X -0.024,Y -396.159,Z 398.446,A 0.000,B 0.000,C 90.000,E1 80.330} C_DIS
LIN {X 0.080,Y -384.316,Z 398.434,A 0.000,B 0.000,C 90.000,E1 78.049} C_DIS
LIN {X -0.014,Y -371.242,Z 398.419,A 0.000,B 0.000,C 90.000,E1 75.463} C_DIS
LIN {X 0.116,Y -359.850,Z 398.406,A 0.000,B 0.000,C 90.000,E1 73.087} C_DIS
LIN {X -0.124,Y -347.542,Z 398.391,A 0.000,B 0.000,C 90.000,E1 70.423} C_DIS
LIN {X -0.123,Y -336.928,Z 398.378,A 0.000,B 0.000,C 90.000,E1 67.975} C_DIS
LIN {X -0.035,Y -325.394,Z 398.362,A 0.000,B 0.000,C 90.000,E1 65.153} C_DIS
LIN {X 0.017,Y -314.486,Z 398.346,A 0.000,B 0.000,C 90.000,E1 62.281} C_DIS
LIN {X -0.157,Y -301.868,Z 398.326,A 0.000,B 0.000,C 90.000,E1 58.742} C_DIS
LIN {X 0.052,Y -290.304,Z 398.306,A 0.000,B 0.000,C 90.000,E1 55.055} C_DIS
LIN {X 0.076,Y -282.601,Z 398.291,A 0.000,B 0.000,C 90.000,E1 52.351} C_DIS
LIN {X 0.030,Y -275.190,Z 398.276,A 0.000,B 0.000,C 90.000,E1 49.622} C_DIS
LIN {X -0.011,Y -269.552,Z 398.264,A 0.000,B 0.000,C 90.000,E1 47.553} C_DIS
LIN {X 0.021,Y -263.687,Z 398.253,A 0.000,B 0.000,C 90.000,E1 45.445} C_DIS
LIN {X -0.057,Y -257.723,Z 398.241,A 0.000,B 0.000,C 90.000,E1 43.338} C_DIS
LIN {X 0.123,Y -251.654,Z 398.229,A 0.000,B 0.000,C 90.000,E1 41.148} C_DIS
LIN {X 0.042,Y -245.508,Z 398.217,A 0.000,B 0.000,C 90.000,E1 38.991} C_DIS
LIN {X -0.129,Y -237.547,Z 398.200,A 0.000,B 0.000,C 90.000,E1 36.091} C_DIS
LIN {X -0.064,Y -230.007,Z 398.184,A 0.000,B 0.000,C 90.000,E1 33.086} C_DIS
LIN {X -0.060,Y -223.032,Z 398.167,A 0.000,B 0.000,C 90.000,E1 30.050} C_DIS
LIN {X 0.023,Y -216.629,Z 398.150,A 0.000,B 0.000,C 90.000,E1 26.950} C_DIS
LIN {X 0.044,Y -210.916,Z 398.132,A 0.000,B 0.000,C 90.000,E1 23.823} C_DIS
LIN {X 0.047,Y -205.826,Z 398.115,A 0.000,B 0.000,C 90.000,E1 20.663} C_DIS
LIN {X 0.010,Y -200.280,Z 398.093,A 0.000,B 0.000,C 90.000,E1 16.677} C_DIS
LIN {X -0.035,Y -195.728,Z 398.070,A 0.000,B 0.000,C 90.000,E1 12.647} C_DIS
LIN {X -0.046,Y -192.171,Z 398.048,A 0.000,B 0.000,C 90.000,E1 8.568} C_DIS
LIN {X -0.061,Y -189.165,Z 398.016,A 0.000,B 0.000,C 90.000,E1 2.808} C_DIS
LIN {X -0.034,Y -188.999,Z 397.965,A 0.000,B 0.000,C 90.000,E1 353.742} C_DIS
LIN {X 0.032,Y -191.520,Z 397.933,A 0.000,B 0.000,C 90.000,E1 347.937} C_DIS
LIN {X 0.012,Y -195.102,Z 397.906,A 0.000,B 0.000,C 90.000,E1 343.015} C_DIS
LIN {X -0.034,Y -199.284,Z 397.883,A 0.000,B 0.000,C 90.000,E1 338.954} C_DIS
LIN {X -0.040,Y -204.560,Z 397.861,A 0.000,B 0.000,C 90.000,E1 334.921} C_DIS
LIN {X -0.001,Y -210.876,Z 397.838,A 0.000,B 0.000,C 90.000,E1 330.923} C_DIS
LIN {X -0.006,Y -217.831,Z 397.817,A 0.000,B 0.000,C 90.000,E1 326.993} C_DIS
LIN {X -0.045,Y -225.436,Z 397.795,A 0.000,B 0.000,C 90.000,E1 323.130} C_DIS
LIN {X 0.037,Y -233.908,Z 397.774,A 0.000,B 0.000,C 90.000,E1 319.299} C_DIS
LIN {X -0.146,Y -242.518,Z 397.755,A 0.000,B 0.000,C 90.000,E1 315.972} C_DIS
LIN {X -0.074,Y -251.200,Z 397.739,A 0.000,B 0.000,C 90.000,E1 313.014} C_DIS
LIN {X 0.074,Y -260.925,Z 397.723,A 0.000,B 0.000,C 90.000,E1 310.092} C_DIS
LIN {X 0.102,Y -270.124,Z 397.709,A 0.000,B 0.000,C 90.000,E1 307.604} C_DIS
LIN {X 0.176,Y -283.893,Z 397.690,A 0.000,B 0.000,C 90.000,E1 304.119} C_DIS
LIN {X -0.119,Y -298.563,Z 397.671,A 0.000,B 0.000,C 90.000,E1 300.797} C_DIS
LIN {X -0.135,Y -309.783,Z 397.658,A 0.000,B 0.000,C 90.000,E1 298.487} C_DIS
LIN {X 0.103,Y -325.858,Z 397.642,A 0.000,B 0.000,C 90.000,E1 295.540} C_DIS
LIN {X 0.148,Y -337.763,Z 397.632,A 0.000,B 0.000,C 90.000,E1 293.643} C_DIS
LIN {X -0.084,Y -357.171,Z 397.616,A 0.000,B 0.000,C 90.000,E1 290.918} C_DIS
LIN {X -0.039,Y -378.114,Z 397.601,A 0.000,B 0.000,C 90.000,E1 288.236} C_DIS
LIN {X -0.159,Y -395.818,Z 397.590,A 0.000,B 0.000,C 90.000,E1 286.260} C_DIS
LIN {X -0.128,Y -419.044,Z 397.577,A 0.000,B 0.000,C 90.000,E1 283.883} C_DIS
LIN {X -0.109,Y -431.932,Z 397.570,A 0.000,B 0.000,C 90.000,E1 282.591} C_DIS
LIN {X -0.176,Y -439.459,Z 397.566,A 0.000,B 0.000,C 90.000,E1 281.827} C_DIS
LIN {X 0.092,Y -446.566,Z 397.561,A 0.000,B 0.000,C 90.000,E1 281.007} C_DIS
LIN {X -0.173,Y -453.177,Z 397.557,A 0.000,B 0.000,C 90.000,E1 280.254} C_DIS
LIN {X 0.079,Y -459.224,Z 397.553,A 0.000,B 0.000,C 90.000,E1 279.443} C_DIS
LIN {X -0.236,Y -466.584,Z 397.547,A 0.000,B 0.000,C 90.000,E1 278.454} C_DIS
LIN {X -0.012,Y -473.297,Z 397.541,A 0.000,B 0.000,C 90.000,E1 277.409} C_DIS
LIN {X 0.233,Y -479.363,Z 397.536,A 0.000,B 0.000,C 90.000,E1 276.372} C_DIS
LIN {X 0.200,Y -483.293,Z 397.531,A 0.000,B 0.000,C 90.000,E1 275.625} C_DIS
LIN {X -0.106,Y -485.539,Z 397.529,A 0.000,B 0.000,C 90.000,E1 275.163} C_DIS
LIN {X 0.081,Y -487.398,Z 397.526,A 0.000,B 0.000,C 90.000,E1 274.645} C_DIS
LIN {X -0.248,Y -488.861,Z 397.523,A 0.000,B 0.000,C 90.000,E1 274.188} C_DIS
LIN {X -0.043,Y -489.981,Z 397.520,A 0.000,B 0.000,C 90.000,E1 273.669} C_DIS
LIN {X 0.139,Y -490.783,Z 397.518,A 0.000,B 0.000,C 90.000,E1 273.154} C_DIS
LIN {X -0.135,Y -491.296,Z 397.515,A 0.000,B 0.000,C 90.000,E1 272.694} C_DIS
LIN {X 0.063,Y -491.490,Z 397.512,A 0.000,B 0.000,C 90.000,E1 272.178} C_DIS
LIN {X -0.210,Y -491.334,Z 397.509,A 0.000,B 0.000,C 90.000,E1 271.718} C_DIS
LIN {X -0.009,Y -490.812,Z 397.507,A 0.000,B 0.000,C 90.000,E1 271.203} C_DIS
LIN {X 0.194,Y -489.896,Z 397.504,A 0.000,B 0.000,C 90.000,E1 270.688} C_DIS
LIN {X -0.095,Y -488.494,Z 397.501,A 0.000,B 0.000,C 90.000,E1 270.229} C_DIS
LIN {X 0.099,Y -486.536,Z 397.498,A 0.000,B 0.000,C 90.000,E1 269.714} C_DIS
LIN {X -0.201,Y -483.898,Z 397.496,A 0.000,B 0.000,C 90.000,E1 269.255} C_DIS
LIN {X -0.035,Y -480.498,Z 397.493,A 0.000,B 0.000,C 90.000,E1 268.740} C_DIS
LIN {X 0.111,Y -476.131,Z 397.490,A 0.000,B 0.000,C 90.000,E1 268.224} C_DIS
LIN {X -0.049,Y -473.492,Z 397.489,A 0.000,B 0.000,C 90.000,E1 267.993} C_DIS
LIN {X -0.132,Y -467.506,Z 397.486,A 0.000,B 0.000,C 90.000,E1 267.535} C_DIS
LIN {X -0.042,Y -464.165,Z 397.485,A 0.000,B 0.000,C 90.000,E1 267.306} C_DIS
LIN {X 0.212,Y -457.206,Z 397.483,A 0.000,B 0.000,C 90.000,E1 266.906} C_DIS
LIN {X 0.148,Y -450.190,Z 397.481,A 0.000,B 0.000,C 90.000,E1 266.617} C_DIS
LIN {X 0.031,Y -442.912,Z 397.480,A 0.000,B 0.000,C 90.000,E1 266.388} C_DIS
LIN {X -0.204,Y -434.686,Z 397.479,A 0.000,B 0.000,C 90.000,E1 266.216} C_DIS
LIN {X 0.013,Y -425.995,Z 397.478,A 0.000,B 0.000,C 90.000,E1 266.045} C_DIS
LIN {X -0.111,Y -418.744,Z 397.478,A 0.000,B 0.000,C 90.000,E1 265.988} C_DIS
LIN {X 0.044,Y -411.010,Z 397.477,A 0.000,B 0.000,C 90.000,E1 265.927} C_DIS
LIN {X -0.005,Y -180.917,Z 397.477,A 0.000,B 0.000,C 90.000,E1 265.927} C_DIS
LIN {X -0.066,Y -180.871,Z 397.472,A 0.000,B 0.000,C 90.000,E1 265.065} C_DIS
LIN {X -0.009,Y -178.988,Z 397.444,A 0.000,B 0.000,C 90.000,E1 259.982} C_DIS
LIN {X 0.003,Y -177.967,Z 397.435,A 0.000,B 0.000,C 90.000,E1 258.285} C_DIS
LIN {X 0.021,Y -175.611,Z 397.411,A 0.000,B 0.000,C 90.000,E1 254.031} C_DIS
LIN {X 0.034,Y -172.333,Z 397.388,A 0.000,B 0.000,C 90.000,E1 249.752} C_DIS
LIN {X 0.013,Y -171.810,Z 397.383,A 0.000,B 0.000,C 90.000,E1 248.901} C_DIS
LIN {X 0.019,Y -170.272,Z 397.373,A 0.000,B 0.000,C 90.000,E1 247.177} C_DIS
LIN {X -0.044,Y -166.813,Z 397.349,A 0.000,B 0.000,C 90.000,E1 242.871} C_DIS
LIN {X 0.013,Y -162.795,Z 397.325,A 0.000,B 0.000,C 90.000,E1 238.486} C_DIS
LIN {X 0.074,Y -161.483,Z 397.315,A 0.000,B 0.000,C 90.000,E1 236.707} C_DIS
LIN {X -0.011,Y -157.478,Z 397.291,A 0.000,B 0.000,C 90.000,E1 232.316} C_DIS
LIN {X 0.046,Y -155.495,Z 397.276,A 0.000,B 0.000,C 90.000,E1 229.622} C_DIS
LIN {X -0.021,Y -151.800,Z 397.251,A 0.000,B 0.000,C 90.000,E1 225.162} C_DIS
LIN {X -0.009,Y -150.011,Z 397.236,A 0.000,B 0.000,C 90.000,E1 222.447} C_DIS
LIN {X 0.022,Y -146.836,Z 397.211,A 0.000,B 0.000,C 90.000,E1 217.890} C_DIS
LIN {X 0.009,Y -145.418,Z 397.195,A 0.000,B 0.000,C 90.000,E1 215.152} C_DIS
LIN {X 0.044,Y -142.845,Z 397.170,A 0.000,B 0.000,C 90.000,E1 210.541} C_DIS
LIN {X -0.026,Y -141.459,Z 397.149,A 0.000,B 0.000,C 90.000,E1 206.873} C_DIS
LIN {X 0.013,Y -139.375,Z 397.113,A 0.000,B 0.000,C 90.000,E1 200.355} C_DIS
LIN {X -0.044,Y -138.824,Z 397.098,A 0.000,B 0.000,C 90.000,E1 197.583} C_DIS
LIN {X 0.044,Y -138.353,Z 397.056,A 0.000,B 0.000,C 90.000,E1 190.074} C_DIS
LIN {X 0.017,Y -139.531,Z 397.004,A 0.000,B 0.000,C 90.000,E1 180.745} C_DIS
LIN {X -0.030,Y -141.210,Z 396.973,A 0.000,B 0.000,C 90.000,E1 175.179} C_DIS
LIN {X 0.071,Y -142.585,Z 396.958,A 0.000,B 0.000,C 90.000,E1 172.356} C_DIS
LIN {X 0.025,Y -144.882,Z 396.932,A 0.000,B 0.000,C 90.000,E1 167.757} C_DIS
LIN {X -0.022,Y -147.508,Z 396.912,A 0.000,B 0.000,C 90.000,E1 164.102} C_DIS
LIN {X 0.053,Y -150.101,Z 396.891,A 0.000,B 0.000,C 90.000,E1 160.423} C_DIS
LIN {X 0.066,Y -153.458,Z 396.871,A 0.000,B 0.000,C 90.000,E1 156.794} C_DIS
LIN {X -0.083,Y -157.822,Z 396.846,A 0.000,B 0.000,C 90.000,E1 152.359} C_DIS
LIN {X -0.051,Y -162.104,Z 396.827,A 0.000,B 0.000,C 90.000,E1 148.791} C_DIS
LIN {X -0.027,Y -166.304,Z 396.807,A 0.000,B 0.000,C 90.000,E1 145.261} C_DIS
LIN {X -0.031,Y -171.322,Z 396.788,A 0.000,B 0.000,C 90.000,E1 141.778} C_DIS
LIN {X 0.004,Y -176.222,Z 396.768,A 0.000,B 0.000,C 90.000,E1 138.324} C_DIS
LIN {X -0.003,Y -180.500,Z 396.754,A 0.000,B 0.000,C 90.000,E1 135.769} C_DIS
LIN {X -0.021,Y -185.903,Z 396.736,A 0.000,B 0.000,C 90.000,E1 132.405} C_DIS
LIN {X 0.040,Y -190.532,Z 396.722,A 0.000,B 0.000,C 90.000,E1 129.886} C_DIS
LIN {X 0.040,Y -197.644,Z 396.699,A 0.000,B 0.000,C 90.000,E1 125.884} C_DIS
LIN {X 0.058,Y -197.790,Z 396.699,A 0.000,B 0.000,C 90.000,E1 125.804} C_DIS
LIN {X 0.052,Y -297.205,Z 396.699,A 0.000,B 0.000,C 90.000,E1 125.804} C_DIS
LIN {X -0.088,Y -298.720,Z 396.699,A 0.000,B 0.000,C 90.000,E1 125.804} C_DIS
LIN {X -0.086,Y -301.848,Z 396.698,A 0.000,B 0.000,C 90.000,E1 125.678} C_DIS
LIN {X 0.095,Y -305.229,Z 396.697,A 0.000,B 0.000,C 90.000,E1 125.391} C_DIS
LIN {X 0.107,Y -308.898,Z 396.694,A 0.000,B 0.000,C 90.000,E1 124.945} C_DIS
LIN {X 0.154,Y -310.783,Z 396.692,A 0.000,B 0.000,C 90.000,E1 124.612} C_DIS
LIN {X -0.054,Y -312.258,Z 396.691,A 0.000,B 0.000,C 90.000,E1 124.326} C_DIS
LIN {X -0.102,Y -324.622,Z 396.671,A 0.000,B 0.000,C 90.000,E1 120.797} C_DIS
LIN {X -0.189,Y -336.114,Z 396.655,A 0.000,B 0.000,C 90.000,E1 117.975} C_DIS
LIN {X 0.051,Y -349.047,Z 396.640,A 0.000,B 0.000,C 90.000,E1 115.155} C_DIS
LIN {X -0.159,Y -361.854,Z 396.626,A 0.000,B 0.000,C 90.000,E1 112.770} C_DIS
LIN {X 0.013,Y -375.987,Z 396.613,A 0.000,B 0.000,C 90.000,E1 110.375} C_DIS
LIN {X 0.059,Y -391.553,Z 396.600,A 0.000,B 0.000,C 90.000,E1 108.055} C_DIS
LIN {X 0.130,Y -408.664,Z 396.588,A 0.000,B 0.000,C 90.000,E1 105.788} C_DIS
LIN {X 0.126,Y -427.450,Z 396.576,A 0.000,B 0.000,C 90.000,E1 103.592} C_DIS
LIN {X -0.058,Y -447.487,Z 396.564,A 0.000,B 0.000,C 90.000,E1 101.535} C_DIS
LIN {X 0.051,Y -468.094,Z 396.553,A 0.000,B 0.000,C 90.000,E1 99.613} C_DIS
LIN {X -0.021,Y -489.038,Z 396.544,A 0.000,B 0.000,C 90.000,E1 97.871} C_DIS
LIN {X 0.128,Y -490.953,Z 396.543,A 0.000,B 0.000,C 90.000,E1 97.644} C_DIS
LIN {X 0.026,Y -492.666,Z 396.541,A 0.000,B 0.000,C 90.000,E1 97.409} C_DIS
LIN {X -0.142,Y -493.951,Z 396.540,A 0.000,B 0.000,C 90.000,E1 97.182} C_DIS
LIN {X 0.099,Y -495.537,Z 396.537,A 0.000,B 0.000,C 90.000,E1 96.663} C_DIS
LIN {X -0.144,Y -496.051,Z 396.534,A 0.000,B 0.000,C 90.000,E1 96.201} C_DIS
LIN {X 0.113,Y -495.574,Z 396.532,A 0.000,B 0.000,C 90.000,E1 95.682} C_DIS
LIN {X -0.119,Y -494.029,Z 396.529,A 0.000,B 0.000,C 90.000,E1 95.220} C_DIS
LIN {X 0.232,Y -492.770,Z 396.528,A 0.000,B 0.000,C 90.000,E1 94.935} C_DIS
LIN {X -0.012,Y -489.271,Z 396.525,A 0.000,B 0.000,C 90.000,E1 94.473} C_DIS
LIN {X -0.103,Y -481.611,Z 396.519,A 0.000,B 0.000,C 90.000,E1 93.498} C_DIS
LIN {X -0.213,Y -460.007,Z 396.504,A 0.000,B 0.000,C 90.000,E1 90.745} C_DIS
LIN {X -0.081,Y -440.205,Z 396.488,A 0.000,B 0.000,C 90.000,E1 87.879} C_DIS
LIN {X 0.172,Y -418.929,Z 396.469,A 0.000,B 0.000,C 90.000,E1 84.375} C_DIS
LIN {X 0.166,Y -406.649,Z 396.457,A 0.000,B 0.000,C 90.000,E1 82.186} C_DIS
LIN {X 0.119,Y -391.586,Z 396.441,A 0.000,B 0.000,C 90.000,E1 79.398} C_DIS
LIN {X 0.078,Y -381.243,Z 396.430,A 0.000,B 0.000,C 90.000,E1 77.409} C_DIS
LIN {X -0.001,Y -369.704,Z 396.417,A 0.000,B 0.000,C 90.000,E1 75.102} C_DIS
LIN {X 0.095,Y -358.339,Z 396.404,A 0.000,B 0.000,C 90.000,E1 72.725} C_DIS
LIN {X 0.143,Y -346.057,Z 396.389,A 0.000,B 0.000,C 90.000,E1 70.007} C_DIS
LIN {X -0.101,Y -334.135,Z 396.374,A 0.000,B 0.000,C 90.000,E1 67.283} C_DIS
LIN {X -0.046,Y -320.304,Z 396.355,A 0.000,B 0.000,C 90.000,E1 63.819} C_DIS
LIN {X 0.056,Y -308.423,Z 396.337,A 0.000,B 0.000,C 90.000,E1 60.589} C_DIS
LIN {X -0.031,Y -297.352,Z 396.318,A 0.000,B 0.000,C 90.000,E1 57.327} C_DIS
LIN {X -0.030,Y -287.236,Z 396.300,A 0.000,B 0.000,C 90.000,E1 53.989} C_DIS
LIN {X -0.063,Y -277.798,Z 396.281,A 0.000,B 0.000,C 90.000,E1 50.598} C_DIS
LIN {X -0.056,Y -272.222,Z 396.270,A 0.000,B 0.000,C 90.000,E1 48.528} C_DIS
LIN {X 0.036,Y -266.496,Z 396.258,A 0.000,B 0.000,C 90.000,E1 46.419} C_DIS
LIN {X 0.009,Y -260.581,Z 396.246,A 0.000,B 0.000,C 90.000,E1 44.312} C_DIS
LIN {X 0.064,Y -254.625,Z 396.234,A 0.000,B 0.000,C 90.000,E1 42.162} C_DIS
LIN {X 0.013,Y -248.498,Z 396.222,A 0.000,B 0.000,C 90.000,E1 40.011} C_DIS
LIN {X 0.057,Y -240.412,Z 396.206,A 0.000,B 0.000,C 90.000,E1 37.076} C_DIS
LIN {X -0.019,Y -230.873,Z 396.185,A 0.000,B 0.000,C 90.000,E1 33.372} C_DIS
LIN {X 0.011,Y -223.810,Z 396.169,A 0.000,B 0.000,C 90.000,E1 30.335} C_DIS
LIN {X -0.001,Y -215.796,Z 396.147,A 0.000,B 0.000,C 90.000,E1 26.488} C_DIS
LIN {X -0.053,Y -208.829,Z 396.125,A 0.000,B 0.000,C 90.000,E1 22.589} C_DIS
LIN {X 0.019,Y -202.860,Z 396.103,A 0.000,B 0.000,C 90.000,E1 18.598} C_DIS
LIN {X -0.035,Y -197.802,Z 396.081,A 0.000,B 0.000,C 90.000,E1 14.592} C_DIS
LIN {X -0.098,Y -193.691,Z 396.058,A 0.000,B 0.000,C 90.000,E1 10.546} C_DIS
LIN {X -0.042,Y -190.739,Z 396.036,A 0.000,B 0.000,C 90.000,E1 6.429} C_DIS
LIN {X 0.000,Y -188.455,Z 396.000,A 0.000,B 0.000,C 90.000,E1 360.000} C_DIS
LIN {X -0.075,Y -190.126,Z 395.947,A 0.000,B 0.000,C 90.000,E1 350.443} C_DIS
LIN {X 0.040,Y -193.017,Z 395.919,A 0.000,B 0.000,C 90.000,E1 345.463} C_DIS
LIN {X -0.073,Y -196.509,Z 395.897,A 0.000,B 0.000,C 90.000,E1 341.402} C_DIS
LIN {X 0.052,Y -201.129,Z 395.874,A 0.000,B 0.000,C 90.000,E1 337.305} C_DIS
LIN {X -0.018,Y -206.853,Z 395.852,A 0.000,B 0.000,C 90.000,E1 333.307} C_DIS
LIN {X 0.017,Y -213.439,Z 395.830,A 0.000,B 0.000,C 90.000,E1 329.331} C_DIS
LIN {X -0.036,Y -220.717,Z 395.808,A 0.000,B 0.000,C 90.000,E1 325.435} C_DIS
LIN {X -0.037,Y -226.943,Z 395.791,A 0.000,B 0.000,C 90.000,E1 322.351} C_DIS
LIN {X -0.004,Y -233.800,Z 395.774,A 0.000,B 0.000,C 90.000,E1 319.299} C_DIS
LIN {X 0.150,Y -242.429,Z 395.755,A 0.000,B 0.000,C 90.000,E1 315.891} C_DIS
LIN {X 0.047,Y -251.123,Z 395.739,A 0.000,B 0.000,C 90.000,E1 312.975} C_DIS
LIN {X 0.019,Y -260.840,Z 395.723,A 0.000,B 0.000,C 90.000,E1 310.092} C_DIS
LIN {X -0.025,Y -268.707,Z 395.711,A 0.000,B 0.000,C 90.000,E1 307.971} C_DIS
LIN {X 0.051,Y -280.979,Z 395.693,A 0.000,B 0.000,C 90.000,E1 304.818} C_DIS
LIN {X 0.069,Y -295.445,Z 395.675,A 0.000,B 0.000,C 90.000,E1 301.416} C_DIS
LIN {X 0.146,Y -306.405,Z 395.662,A 0.000,B 0.000,C 90.000,E1 299.077} C_DIS
LIN {X 0.010,Y -322.150,Z 395.645,A 0.000,B 0.000,C 90.000,E1 296.181} C_DIS
LIN {X 0.119,Y -333.745,Z 395.635,A 0.000,B 0.000,C 90.000,E1 294.259} C_DIS
LIN {X -0.205,Y -355.119,Z 395.618,A 0.000,B 0.000,C 90.000,E1 291.227} C_DIS
LIN {X 0.139,Y -375.892,Z 395.603,A 0.000,B 0.000,C 90.000,E1 288.489} C_DIS
LIN {X -0.186,Y -390.945,Z 395.593,A 0.000,B 0.000,C 90.000,E1 286.804} C_DIS
LIN {X 0.120,Y -411.688,Z 395.581,A 0.000,B 0.000,C 90.000,E1 284.592} C_DIS
LIN {X -0.137,Y -424.522,Z 395.574,A 0.000,B 0.000,C 90.000,E1 283.355} C_DIS
LIN {X 0.051,Y -434.699,Z 395.568,A 0.000,B 0.000,C 90.000,E1 282.299} C_DIS
LIN {X -0.065,Y -442.113,Z 395.564,A 0.000,B 0.000,C 90.000,E1 281.535} C_DIS
LIN {X 0.097,Y -449.000,Z 395.560,A 0.000,B 0.000,C 90.000,E1 280.725} C_DIS
LIN {X -0.055,Y -455.420,Z 395.555,A 0.000,B 0.000,C 90.000,E1 279.962} C_DIS
LIN {X 0.040,Y -463.103,Z 395.550,A 0.000,B 0.000,C 90.000,E1 278.916} C_DIS
LIN {X 0.226,Y -470.131,Z 395.544,A 0.000,B 0.000,C 90.000,E1 277.871} C_DIS
LIN {X -0.039,Y -476.512,Z 395.538,A 0.000,B 0.000,C 90.000,E1 276.891} C_DIS
LIN {X -0.100,Y -480.805,Z 395.534,A 0.000,B 0.000,C 90.000,E1 276.144} C_DIS
LIN {X -0.069,Y -484.538,Z 395.530,A 0.000,B 0.000,C 90.000,E1 275.391} C_DIS
LIN {X -0.058,Y -487.436,Z 395.526,A 0.000,B 0.000,C 90.000,E1 274.645} C_DIS
LIN {X 0.099,Y -488.889,Z 395.523,A 0.000,B 0.000,C 90.000,E1 274.131} C_DIS
LIN {X -0.185,Y -489.980,Z 395.520,A 0.000,B 0.000,C 90.000,E1 273.669} C_DIS
LIN {X -0.002,Y -490.752,Z 395.518,A 0.000,B 0.000,C 90.000,E1 273.154} C_DIS
LIN {X 0.216,Y -491.259,Z 395.515,A 0.000,B 0.000,C 90.000,E1 272.636} C_DIS
LIN {X -0.079,Y -491.455,Z 395.512,A 0.000,B 0.000,C 90.000,E1 272.178} C_DIS
LIN {X 0.139,Y -491.303,Z 395.509,A 0.000,B 0.000,C 90.000,E1 271.661} C_DIS
LIN {X -0.150,Y -490.772,Z 395.507,A 0.000,B 0.000,C 90.000,E1 271.203} C_DIS
LIN {X 0.052,Y -489.833,Z 395.504,A 0.000,B 0.000,C 90.000,E1 270.688} C_DIS
LIN {X -0.237,Y -488.427,Z 395.501,A 0.000,B 0.000,C 90.000,E1 270.229} C_DIS
LIN {X -0.042,Y -486.464,Z 395.498,A 0.000,B 0.000,C 90.000,E1 269.714} C_DIS
LIN {X 0.143,Y -483.804,Z 395.496,A 0.000,B 0.000,C 90.000,E1 269.198} C_DIS
LIN {X -0.016,Y -482.234,Z 395.494,A 0.000,B 0.000,C 90.000,E1 268.969} C_DIS
LIN {X 0.138,Y -478.318,Z 395.491,A 0.000,B 0.000,C 90.000,E1 268.453} C_DIS
LIN {X -0.188,Y -473.323,Z 395.489,A 0.000,B 0.000,C 90.000,E1 267.993} C_DIS
LIN {X 0.207,Y -467.290,Z 395.486,A 0.000,B 0.000,C 90.000,E1 267.478} C_DIS
LIN {X -0.162,Y -463.952,Z 395.485,A 0.000,B 0.000,C 90.000,E1 267.306} C_DIS
LIN {X 0.102,Y -456.981,Z 395.483,A 0.000,B 0.000,C 90.000,E1 266.906} C_DIS
LIN {X 0.062,Y -450.038,Z 395.481,A 0.000,B 0.000,C 90.000,E1 266.617} C_DIS
LIN {X -0.049,Y -442.720,Z 395.480,A 0.000,B 0.000,C 90.000,E1 266.388} C_DIS
LIN {X 0.180,Y -434.518,Z 395.479,A 0.000,B 0.000,C 90.000,E1 266.159} C_DIS
LIN {X -0.020,Y -426.061,Z 395.478,A 0.000,B 0.000,C 90.000,E1 266.045} C_DIS
LIN {X -0.150,Y -418.723,Z 395.478,A 0.000,B 0.000,C 90.000,E1 265.988} C_DIS
LIN {X 0.006,Y -409.893,Z 395.477,A 0.000,B 0.000,C 90.000,E1 265.927} C_DIS
LIN {X -0.021,Y -180.916,Z 395.477,A 0.000,B 0.000,C 90.000,E1 265.927} C_DIS
LIN {X -0.079,Y -180.870,Z 395.472,A 0.000,B 0.000,C 90.000,E1 265.065} C_DIS
LIN {X -0.022,Y -178.986,Z 395.444,A 0.000,B 0.000,C 90.000,E1 259.982} C_DIS
LIN {X -0.010,Y -177.965,Z 395.435,A 0.000,B 0.000,C 90.000,E1 258.285} C_DIS
LIN {X 0.008,Y -175.607,Z 395.411,A 0.000,B 0.000,C 90.000,E1 254.031} C_DIS
LIN {X 0.021,Y -172.331,Z 395.388,A 0.000,B 0.000,C 90.000,E1 249.752} C_DIS
LIN {X 0.000,Y -171.807,Z 395.383,A 0.000,B 0.000,C 90.000,E1 248.901} C_DIS
LIN {X 0.007,Y -170.269,Z 395.373,A 0.000,B 0.000,C 90.000,E1 247.177} C_DIS
LIN {X -0.057,Y -166.811,Z 395.349,A 0.000,B 0.000,C 90.000,E1 242.871} C_DIS
LIN {X 0.001,Y -162.792,Z 395.325,A 0.000,B 0.000,C 90.000,E1 238.486} C_DIS
LIN {X 0.061,Y -161.480,Z 395.315,A 0.000,B 0.000,C 90.000,E1 236.707} C_DIS
LIN {X -0.023,Y -157.475,Z 395.291,A 0.000,B 0.000,C 90.000,E1 232.316} C_DIS
LIN {X 0.034,Y -155.490,Z 395.276,A 0.000,B 0.000,C 90.000,E1 229.622} C_DIS
LIN {X -0.034,Y -151.797,Z 395.251,A 0.000,B 0.000,C 90.000,E1 225.162} C_DIS
LIN {X -0.020,Y -150.007,Z 395.236,A 0.000,B 0.000,C 90.000,E1 222.447} C_DIS
LIN {X 0.011,Y -146.833,Z 395.211,A 0.000,B 0.000,C 90.000,E1 217.890} C_DIS
LIN {X -0.003,Y -145.414,Z 395.195,A 0.000,B 0.000,C 90.000,E1 215.152} C_DIS
LIN {X 0.033,Y -142.843,Z 395.170,A 0.000,B 0.000,C 90.000,E1 210.541} C_DIS
LIN {X -0.038,Y -141.457,Z 395.149,A 0.000,B 0.000,C 90.000,E1 206.873} C_DIS
LIN {X 0.002,Y -139.374,Z 395.113,A 0.000,B 0.000,C 90.000,E1 200.355} C_DIS
LIN {X -0.056,Y -138.824,Z 395.098,A 0.000,B 0.000,C 90.000,E1 197.583} C_DIS
LIN {X 0.033,Y -138.353,Z 395.056,A 0.000,B 0.000,C 90.000,E1 190.074} C_DIS
LIN {X 0.006,Y -139.532,Z 395.004,A 0.000,B 0.000,C 90.000,E1 180.745} C_DIS
LIN {X -0.041,Y -141.212,Z 394.973,A 0.000,B 0.000,C 90.000,E1 175.179} C_DIS
LIN {X 0.059,Y -142.586,Z 394.958,A 0.000,B 0.000,C 90.000,E1 172.356} C_DIS
LIN {X 0.013,Y -144.884,Z 394.932,A 0.000,B 0.000,C 90.000,E1 167.757} C_DIS
LIN {X -0.034,Y -147.512,Z 394.912,A 0.000,B 0.000,C 90.000,E1 164.102} C_DIS
LIN {X 0.041,Y -150.105,Z 394.891,A 0.000,B 0.000,C 90.000,E1 160.423} C_DIS
LIN {X 0.054,Y -153.462,Z 394.871,A 0.000,B 0.000,C 90.000,E1 156.794} C_DIS
LIN {X -0.095,Y -157.826,Z 394.846,A 0.000,B 0.000,C 90.000,E1 152.359} C_DIS
LIN {X 0.076,Y -162.109,Z 394.826,A 0.000,B 0.000,C 90.000,E1 148.742} C_DIS
LIN {X -0.040,Y -166.311,Z 394.807,A 0.000,B 0.000,C 90.000,E1 145.261} C_DIS
LIN {X 0.063,Y -171.327,Z 394.788,A 0.000,B 0.000,C 90.000,E1 141.743} C_DIS
LIN {X -0.009,Y -176.228,Z 394.768,A 0.000,B 0.000,C 90.000,E1 138.324} C_DIS
LIN {X 0.110,Y -180.507,Z 394.754,A 0.000,B 0.000,C 90.000,E1 135.729} C_DIS
LIN {X 0.090,Y -185.911,Z 394.736,A 0.000,B 0.000,C 90.000,E1 132.366} C_DIS
LIN {X 0.026,Y -190.539,Z 394.722,A 0.000,B 0.000,C 90.000,E1 129.886} C_DIS
LIN {X 0.057,Y -196.290,Z 394.703,A 0.000,B 0.000,C 90.000,E1 126.583} C_DIS
LIN {X -0.119,Y -197.891,Z 394.699,A 0.000,B 0.000,C 90.000,E1 125.804} C_DIS
LIN {X 0.027,Y -297.295,Z 394.699,A 0.000,B 0.000,C 90.000,E1 125.758} C_DIS
LIN {X -0.053,Y -299.604,Z 394.698,A 0.000,B 0.000,C 90.000,E1 125.724} C_DIS
LIN {X 0.054,Y -303.286,Z 394.697,A 0.000,B 0.000,C 90.000,E1 125.518} C_DIS
LIN {X 0.162,Y -305.536,Z 394.696,A 0.000,B 0.000,C 90.000,E1 125.311} C_DIS
LIN {X -0.048,Y -308.667,Z 394.694,A 0.000,B 0.000,C 90.000,E1 124.978} C_DIS
LIN {X -0.058,Y -310.619,Z 394.693,A 0.000,B 0.000,C 90.000,E1 124.659} C_DIS
LIN {X 0.010,Y -312.143,Z 394.691,A 0.000,B 0.000,C 90.000,E1 124.326} C_DIS
LIN {X -0.153,Y -314.416,Z 394.687,A 0.000,B 0.000,C 90.000,E1 123.706} C_DIS
LIN {X -0.038,Y -324.559,Z 394.671,A 0.000,B 0.000,C 90.000,E1 120.797} C_DIS
LIN {X -0.125,Y -336.044,Z 394.655,A 0.000,B 0.000,C 90.000,E1 117.975} C_DIS
LIN {X 0.116,Y -348.971,Z 394.640,A 0.000,B 0.000,C 90.000,E1 115.155} C_DIS
LIN {X -0.093,Y -361.772,Z 394.626,A 0.000,B 0.000,C 90.000,E1 112.770} C_DIS
LIN {X 0.078,Y -375.900,Z 394.613,A 0.000,B 0.000,C 90.000,E1 110.375} C_DIS
LIN {X 0.124,Y -391.458,Z 394.600,A 0.000,B 0.000,C 90.000,E1 108.055} C_DIS
LIN {X -0.197,Y -408.562,Z 394.588,A 0.000,B 0.000,C 90.000,E1 105.843} C_DIS
LIN {X 0.193,Y -427.340,Z 394.576,A 0.000,B 0.000,C 90.000,E1 103.592} C_DIS
LIN {X 0.006,Y -447.374,Z 394.564,A 0.000,B 0.000,C 90.000,E1 101.535} C_DIS
LIN {X 0.111,Y -467.979,Z 394.553,A 0.000,B 0.000,C 90.000,E1 99.613} C_DIS
LIN {X 0.037,Y -488.972,Z 394.544,A 0.000,B 0.000,C 90.000,E1 97.871} C_DIS
LIN {X 0.185,Y -490.949,Z 394.543,A 0.000,B 0.000,C 90.000,E1 97.644} C_DIS
LIN {X 0.082,Y -492.712,Z 394.541,A 0.000,B 0.000,C 90.000,E1 97.409} C_DIS
LIN {X -0.085,Y -494.033,Z 394.540,A 0.000,B 0.000,C 90.000,E1 97.182} C_DIS
LIN {X 0.157,Y -495.673,Z 394.537,A 0.000,B 0.000,C 90.000,E1 96.663} C_DIS
LIN {X -0.086,Y -496.231,Z 394.534,A 0.000,B 0.000,C 90.000,E1 96.201} C_DIS
LIN {X 0.173,Y -495.798,Z 394.532,A 0.000,B 0.000,C 90.000,E1 95.682} C_DIS
LIN {X -0.060,Y -494.305,Z 394.529,A 0.000,B 0.000,C 90.000,E1 95.220} C_DIS
LIN {X -0.200,Y -493.080,Z 394.528,A 0.000,B 0.000,C 90.000,E1 94.992} C_DIS
LIN {X 0.049,Y -489.644,Z 394.525,A 0.000,B 0.000,C 90.000,E1 94.473} C_DIS
LIN {X -0.039,Y -481.998,Z 394.519,A 0.000,B 0.000,C 90.000,E1 93.498} C_DIS
LIN {X -0.140,Y -460.385,Z 394.504,A 0.000,B 0.000,C 90.000,E1 90.745} C_DIS
LIN {X 0.000,Y -440.544,Z 394.488,A 0.000,B 0.000,C 90.000,E1 87.879} C_DIS
LIN {X -0.157,Y -419.231,Z 394.469,A 0.000,B 0.000,C 90.000,E1 84.432} C_DIS
LIN {X 0.200,Y -408.481,Z 394.458,A 0.000,B 0.000,C 90.000,E1 82.470} C_DIS
LIN {X 0.148,Y -393.396,Z 394.443,A 0.000,B 0.000,C 90.000,E1 79.690} C_DIS
LIN {X 0.147,Y -383.078,Z 394.432,A 0.000,B 0.000,C 90.000,E1 77.701} C_DIS
LIN {X 0.107,Y -370.037,Z 394.417,A 0.000,B 0.000,C 90.000,E1 75.102} C_DIS
LIN {X -0.135,Y -358.645,Z 394.404,A 0.000,B 0.000,C 90.000,E1 72.779} C_DIS
LIN {X -0.066,Y -346.307,Z 394.389,A 0.000,B 0.000,C 90.000,E1 70.061} C_DIS
LIN {X 0.017,Y -334.332,Z 394.374,A 0.000,B 0.000,C 90.000,E1 67.283} C_DIS
LIN {X -0.067,Y -320.455,Z 394.355,A 0.000,B 0.000,C 90.000,E1 63.845} C_DIS
LIN {X 0.070,Y -307.448,Z 394.335,A 0.000,B 0.000,C 90.000,E1 60.284} C_DIS
LIN {X -0.132,Y -295.385,Z 394.315,A 0.000,B 0.000,C 90.000,E1 56.707} C_DIS
LIN {X -0.019,Y -285.427,Z 394.296,A 0.000,B 0.000,C 90.000,E1 53.336} C_DIS
LIN {X 0.056,Y -277.914,Z 394.281,A 0.000,B 0.000,C 90.000,E1 50.598} C_DIS
LIN {X 0.064,Y -272.335,Z 394.270,A 0.000,B 0.000,C 90.000,E1 48.528} C_DIS
LIN {X -0.029,Y -266.647,Z 394.258,A 0.000,B 0.000,C 90.000,E1 46.458} C_DIS
LIN {X -0.055,Y -260.759,Z 394.246,A 0.000,B 0.000,C 90.000,E1 44.352} C_DIS
LIN {X -0.005,Y -254.815,Z 394.234,A 0.000,B 0.000,C 90.000,E1 42.204} C_DIS
LIN {X 0.133,Y -248.702,Z 394.222,A 0.000,B 0.000,C 90.000,E1 40.011} C_DIS
LIN {X 0.033,Y -240.623,Z 394.206,A 0.000,B 0.000,C 90.000,E1 37.111} C_DIS
LIN {X 0.104,Y -231.080,Z 394.186,A 0.000,B 0.000,C 90.000,E1 33.372} C_DIS
LIN {X -0.058,Y -223.999,Z 394.169,A 0.000,B 0.000,C 90.000,E1 30.384} C_DIS
LIN {X -0.044,Y -217.484,Z 394.152,A 0.000,B 0.000,C 90.000,E1 27.308} C_DIS
LIN {X -0.095,Y -211.649,Z 394.134,A 0.000,B 0.000,C 90.000,E1 24.207} C_DIS
LIN {X -0.066,Y -206.414,Z 394.117,A 0.000,B 0.000,C 90.000,E1 21.046} C_DIS
LIN {X -0.013,Y -200.748,Z 394.095,A 0.000,B 0.000,C 90.000,E1 17.040} C_DIS
LIN {X -0.038,Y -196.052,Z 394.072,A 0.000,B 0.000,C 90.000,E1 13.008} C_DIS
LIN {X 0.000,Y -192.301,Z 394.050,A 0.000,B 0.000,C 90.000,E1 8.916} C_DIS
LIN {X 0.079,Y -189.442,Z 394.022,A 0.000,B 0.000,C 90.000,E1 3.955} C_DIS
LIN {X -0.041,Y -188.803,Z 393.965,A 0.000,B 0.000,C 90.000,E1 353.742} C_DIS
LIN {X 0.016,Y -191.293,Z 393.933,A 0.000,B 0.000,C 90.000,E1 347.937} C_DIS
LIN {X -0.013,Y -194.854,Z 393.906,A 0.000,B 0.000,C 90.000,E1 343.015} C_DIS
LIN {X -0.068,Y -198.992,Z 393.883,A 0.000,B 0.000,C 90.000,E1 338.954} C_DIS
LIN {X -0.084,Y -204.312,Z 393.861,A 0.000,B 0.000,C 90.000,E1 334.921} C_DIS
LIN {X 0.038,Y -209.249,Z 393.843,A 0.000,B 0.000,C 90.000,E1 331.691} C_DIS
LIN {X 0.064,Y -216.150,Z 393.821,A 0.000,B 0.000,C 90.000,E1 327.740} C_DIS
LIN {X 0.001,Y -222.100,Z 393.804,A 0.000,B 0.000,C 90.000,E1 324.642} C_DIS
LIN {X 0.006,Y -230.173,Z 393.782,A 0.000,B 0.000,C 90.000,E1 320.803} C_DIS
LIN {X -0.058,Y -237.374,Z 393.765,A 0.000,B 0.000,C 90.000,E1 317.796} C_DIS
LIN {X 0.026,Y -246.565,Z 393.747,A 0.000,B 0.000,C 90.000,E1 314.433} C_DIS
LIN {X 0.058,Y -256.973,Z 393.729,A 0.000,B 0.000,C 90.000,E1 311.148} C_DIS
LIN {X 0.017,Y -267.334,Z 393.713,A 0.000,B 0.000,C 90.000,E1 308.302} C_DIS
LIN {X 0.049,Y -279.468,Z 393.695,A 0.000,B 0.000,C 90.000,E1 305.152} C_DIS
LIN {X 0.024,Y -292.362,Z 393.678,A 0.000,B 0.000,C 90.000,E1 302.084} C_DIS
LIN {X 0.048,Y -304.723,Z 393.663,A 0.000,B 0.000,C 90.000,E1 299.411} C_DIS
LIN {X 0.008,Y -320.310,Z 393.647,A 0.000,B 0.000,C 90.000,E1 296.488} C_DIS
LIN {X -0.018,Y -329.790,Z 393.638,A 0.000,B 0.000,C 90.000,E1 294.899} C_DIS
LIN {X 0.119,Y -350.869,Z 393.621,A 0.000,B 0.000,C 90.000,E1 291.770} C_DIS
LIN {X 0.080,Y -373.701,Z 393.604,A 0.000,B 0.000,C 90.000,E1 288.779} C_DIS
LIN {X -0.085,Y -390.963,Z 393.593,A 0.000,B 0.000,C 90.000,E1 286.804} C_DIS
LIN {X -0.099,Y -411.612,Z 393.581,A 0.000,B 0.000,C 90.000,E1 284.647} C_DIS
LIN {X 0.039,Y -424.439,Z 393.574,A 0.000,B 0.000,C 90.000,E1 283.355} C_DIS
LIN {X -0.121,Y -434.523,Z 393.569,A 0.000,B 0.000,C 90.000,E1 282.355} C_DIS
LIN {X 0.186,Y -441.891,Z 393.564,A 0.000,B 0.000,C 90.000,E1 281.535} C_DIS
LIN {X -0.105,Y -448.789,Z 393.560,A 0.000,B 0.000,C 90.000,E1 280.782} C_DIS
LIN {X 0.186,Y -455.198,Z 393.555,A 0.000,B 0.000,C 90.000,E1 279.962} C_DIS
LIN {X -0.175,Y -462.901,Z 393.550,A 0.000,B 0.000,C 90.000,E1 278.973} C_DIS
LIN {X -0.060,Y -469.934,Z 393.544,A 0.000,B 0.000,C 90.000,E1 277.936} C_DIS
LIN {X 0.206,Y -476.320,Z 393.538,A 0.000,B 0.000,C 90.000,E1 276.891} C_DIS
LIN {X 0.145,Y -480.610,Z 393.534,A 0.000,B 0.000,C 90.000,E1 276.144} C_DIS
LIN {X 0.176,Y -484.371,Z 393.530,A 0.000,B 0.000,C 90.000,E1 275.391} C_DIS
LIN {X 0.187,Y -487.297,Z 393.526,A 0.000,B 0.000,C 90.000,E1 274.645} C_DIS
LIN {X -0.142,Y -488.771,Z 393.523,A 0.000,B 0.000,C 90.000,E1 274.188} C_DIS
LIN {X 0.061,Y -489.895,Z 393.520,A 0.000,B 0.000,C 90.000,E1 273.669} C_DIS
LIN {X -0.246,Y -490.698,Z 393.518,A 0.000,B 0.000,C 90.000,E1 273.212} C_DIS
LIN {X -0.030,Y -491.225,Z 393.515,A 0.000,B 0.000,C 90.000,E1 272.694} C_DIS
LIN {X 0.166,Y -491.434,Z 393.512,A 0.000,B 0.000,C 90.000,E1 272.178} C_DIS
LIN {X -0.108,Y -491.309,Z 393.509,A 0.000,B 0.000,C 90.000,E1 271.718} C_DIS
LIN {X 0.095,Y -490.791,Z 393.507,A 0.000,B 0.000,C 90.000,E1 271.203} C_DIS
LIN {X -0.193,Y -489.923,Z 393.504,A 0.000,B 0.000,C 90.000,E1 270.745} C_DIS
LIN {X 0.007,Y -488.542,Z 393.501,A 0.000,B 0.000,C 90.000,E1 270.229} C_DIS
LIN {X 0.201,Y -486.625,Z 393.499,A 0.000,B 0.000,C 90.000,E1 269.714} C_DIS
LIN {X -0.099,Y -484.013,Z 393.496,A 0.000,B 0.000,C 90.000,E1 269.255} C_DIS
LIN {X 0.226,Y -482.465,Z 393.494,A 0.000,B 0.000,C 90.000,E1 268.969} C_DIS
LIN {X -0.099,Y -478.616,Z 393.492,A 0.000,B 0.000,C 90.000,E1 268.511} C_DIS
LIN {X 0.212,Y -476.296,Z 393.490,A 0.000,B 0.000,C 90.000,E1 268.224} C_DIS
LIN {X 0.052,Y -473.663,Z 393.489,A 0.000,B 0.000,C 90.000,E1 267.993} C_DIS
LIN {X -0.122,Y -470.716,Z 393.487,A 0.000,B 0.000,C 90.000,E1 267.764} C_DIS
LIN {X -0.068,Y -467.715,Z 393.486,A 0.000,B 0.000,C 90.000,E1 267.535} C_DIS
LIN {X -0.104,Y -461.151,Z 393.484,A 0.000,B 0.000,C 90.000,E1 267.135} C_DIS
LIN {X 0.014,Y -454.276,Z 393.482,A 0.000,B 0.000,C 90.000,E1 266.788} C_DIS
LIN {X 0.121,Y -447.124,Z 393.481,A 0.000,B 0.000,C 90.000,E1 266.502} C_DIS
LIN {X 0.161,Y -439.581,Z 393.479,A 0.000,B 0.000,C 90.000,E1 266.274} C_DIS
LIN {X 0.141,Y -431.525,Z 393.478,A 0.000,B 0.000,C 90.000,E1 266.102} C_DIS
LIN {X 0.049,Y -422.471,Z 393.478,A 0.000,B 0.000,C 90.000,E1 265.988} C_DIS
LIN {X 0.004,Y -411.627,Z 393.477,A 0.000,B 0.000,C 90.000,E1 265.927} C_DIS
LIN {X -0.022,Y -180.917,Z 393.477,A 0.000,B 0.000,C 90.000,E1 265.927} C_DIS
LIN {X -0.081,Y -180.870,Z 393.472,A 0.000,B 0.000,C 90.000,E1 265.065} C_DIS
LIN {X -0.024,Y -178.986,Z 393.444,A 0.000,B 0.000,C 90.000,E1 259.982} C_DIS
LIN {X -0.012,Y -177.964,Z 393.435,A 0.000,B 0.000,C 90.000,E1 258.285} C_DIS
LIN {X 0.007,Y -175.608,Z 393.411,A 0.000,B 0.000,C 90.000,E1 254.031} C_DIS
LIN {X 0.020,Y -172.330,Z 393.388,A 0.000,B 0.000,C 90.000,E1 249.752} C_DIS
LIN {X -0.002,Y -171.807,Z 393.383,A 0.000,B 0.000,C 90.000,E1 248.901} C_DIS
LIN {X 0.006,Y -170.268,Z 393.373,A 0.000,B 0.000,C 90.000,E1 247.177} C_DIS
LIN {X -0.058,Y -166.810,Z 393.349,A 0.000,B 0.000,C 90.000,E1 242.871} C_DIS
LIN {X 0.000,Y -162.792,Z 393.325,A 0.000,B 0.000,C 90.000,E1 238.486} C_DIS
LIN {X 0.060,Y -161.479,Z 393.315,A 0.000,B 0.000,C 90.000,E1 236.707} C_DIS
LIN {X -0.025,Y -157.475,Z 393.291,A 0.000,B 0.000,C 90.000,E1 232.316} C_DIS
LIN {X 0.033,Y -155.490,Z 393.276,A 0.000,B 0.000,C 90.000,E1 229.622} C_DIS
LIN {X -0.035,Y -151.797,Z 393.251,A 0.000,B 0.000,C 90.000,E1 225.162} C_DIS
LIN {X -0.022,Y -150.006,Z 393.236,A 0.000,B 0.000,C 90.000,E1 222.447} C_DIS
LIN {X 0.009,Y -146.833,Z 393.211,A 0.000,B 0.000,C 90.000,E1 217.890} C_DIS
LIN {X -0.004,Y -145.413,Z 393.195,A 0.000,B 0.000,C 90.000,E1 215.152} C_DIS
LIN {X 0.031,Y -142.843,Z 393.170,A 0.000,B 0.000,C 90.000,E1 210.541} C_DIS
LIN {X -0.039,Y -141.457,Z 393.149,A 0.000,B 0.000,C 90.000,E1 206.873} C_DIS
LIN {X 0.001,Y -139.373,Z 393.113,A 0.000,B 0.000,C 90.000,E1 200.355} C_DIS
LIN {X -0.057,Y -138.824,Z 393.098,A 0.000,B 0.000,C 90.000,E1 197.583} C_DIS
LIN {X 0.032,Y -138.353,Z 393.056,A 0.000,B 0.000,C 90.000,E1 190.074} C_DIS
LIN {X 0.005,Y -139.532,Z 393.004,A 0.000,B 0.000,C 90.000,E1 180.745} C_DIS
LIN {X -0.043,Y -141.212,Z 392.973,A 0.000,B 0.000,C 90.000,E1 175.179} C_DIS
LIN {X 0.058,Y -142.586,Z 392.958,A 0.000,B 0.000,C 90.000,E1 172.356} C_DIS
LIN {X 0.012,Y -144.885,Z 392.932,A 0.000,B 0.000,C 90.000,E1 167.757} C_DIS
LIN {X -0.035,Y -147.512,Z 392.912,A 0.000,B 0.000,C 90.000,E1 164.102} C_DIS
LIN {X 0.040,Y -150.106,Z 392.891,A 0.000,B 0.000,C 90.000,E1 160.423} C_DIS
LIN {X 0.052,Y -153.463,Z 392.871,A 0.000,B 0.000,C 90.000,E1 156.794} C_DIS
LIN {X -0.096,Y -157.826,Z 392.846,A 0.000,B 0.000,C 90.000,E1 152.359} C_DIS
LIN {X 0.073,Y -162.110,Z 392.826,A 0.000,B 0.000,C 90.000,E1 148.742} C_DIS
LIN {X -0.040,Y -166.311,Z 392.807,A 0.000,B 0.000,C 90.000,E1 145.261} C_DIS
LIN {X 0.061,Y -171.329,Z 392.788,A 0.000,B 0.000,C 90.000,E1 141.743} C_DIS
LIN {X -0.011,Y -176.229,Z 392.768,A 0.000,B 0.000,C 90.000,E1 138.324} C_DIS
LIN {X 0.109,Y -180.509,Z 392.754,A 0.000,B 0.000,C 90.000,E1 135.729} C_DIS
LIN {X 0.089,Y -185.911,Z 392.736,A 0.000,B 0.000,C 90.000,E1 132.366} C_DIS
LIN {X 0.024,Y -190.539,Z 392.722,A 0.000,B 0.000,C 90.000,E1 129.886} C_DIS
LIN {X 0.055,Y -196.290,Z 392.703,A 0.000,B 0.000,C 90.000,E1 126.583} C_DIS
LIN {X -0.001,Y -197.981,Z 392.698,A 0.000,B 0.000,C 90.000,E1 125.724} C_DIS
LIN {X -0.055,Y -297.254,Z 392.698,A 0.000,B 0.000,C 90.000,E1 125.724} C_DIS
LIN {X 0.051,Y -302.665,Z 392.697,A 0.000,B 0.000,C 90.000,E1 125.518} C_DIS
LIN {X 0.159,Y -305.140,Z 392.696,A 0.000,B 0.000,C 90.000,E1 125.311} C_DIS
LIN {X -0.050,Y -308.455,Z 392.694,A 0.000,B 0.000,C 90.000,E1 124.978} C_DIS
LIN {X 0.009,Y -310.417,Z 392.693,A 0.000,B 0.000,C 90.000,E1 124.659} C_DIS
LIN {X 0.146,Y -311.957,Z 392.691,A 0.000,B 0.000,C 90.000,E1 124.326} C_DIS
LIN {X -0.016,Y -314.314,Z 392.687,A 0.000,B 0.000,C 90.000,E1 123.706} C_DIS
LIN {X 0.101,Y -324.445,Z 392.671,A 0.000,B 0.000,C 90.000,E1 120.797} C_DIS
LIN {X 0.015,Y -335.919,Z 392.655,A 0.000,B 0.000,C 90.000,E1 117.975} C_DIS
LIN {X -0.058,Y -348.833,Z 392.640,A 0.000,B 0.000,C 90.000,E1 115.207} C_DIS
LIN {X 0.050,Y -361.620,Z 392.627,A 0.000,B 0.000,C 90.000,E1 112.770} C_DIS
LIN {X -0.130,Y -375.735,Z 392.613,A 0.000,B 0.000,C 90.000,E1 110.429} C_DIS
LIN {X -0.101,Y -391.280,Z 392.601,A 0.000,B 0.000,C 90.000,E1 108.109} C_DIS
LIN {X -0.048,Y -408.369,Z 392.588,A 0.000,B 0.000,C 90.000,E1 105.843} C_DIS
LIN {X -0.071,Y -427.129,Z 392.576,A 0.000,B 0.000,C 90.000,E1 103.647} C_DIS
LIN {X 0.151,Y -447.157,Z 392.564,A 0.000,B 0.000,C 90.000,E1 101.535} C_DIS
LIN {X -0.213,Y -467.757,Z 392.554,A 0.000,B 0.000,C 90.000,E1 99.670} C_DIS
LIN {X 0.167,Y -488.797,Z 392.544,A 0.000,B 0.000,C 90.000,E1 97.871} C_DIS
LIN {X -0.172,Y -490.862,Z 392.543,A 0.000,B 0.000,C 90.000,E1 97.701} C_DIS
LIN {X 0.223,Y -492.684,Z 392.541,A 0.000,B 0.000,C 90.000,E1 97.409} C_DIS
LIN {X 0.066,Y -494.053,Z 392.540,A 0.000,B 0.000,C 90.000,E1 97.182} C_DIS
LIN {X -0.184,Y -495.780,Z 392.537,A 0.000,B 0.000,C 90.000,E1 96.720} C_DIS
LIN {X 0.066,Y -496.412,Z 392.534,A 0.000,B 0.000,C 90.000,E1 96.201} C_DIS
LIN {X -0.168,Y -496.051,Z 392.532,A 0.000,B 0.000,C 90.000,E1 95.739} C_DIS
LIN {X 0.093,Y -494.638,Z 392.529,A 0.000,B 0.000,C 90.000,E1 95.220} C_DIS
LIN {X -0.046,Y -493.463,Z 392.528,A 0.000,B 0.000,C 90.000,E1 94.992} C_DIS
LIN {X 0.203,Y -490.088,Z 392.525,A 0.000,B 0.000,C 90.000,E1 94.473} C_DIS
LIN {X 0.118,Y -482.483,Z 392.520,A 0.000,B 0.000,C 90.000,E1 93.498} C_DIS
LIN {X 0.229,Y -462.742,Z 392.506,A 0.000,B 0.000,C 90.000,E1 90.974} C_DIS
LIN {X -0.014,Y -442.694,Z 392.490,A 0.000,B 0.000,C 90.000,E1 88.165} C_DIS
LIN {X -0.130,Y -421.166,Z 392.471,A 0.000,B 0.000,C 90.000,E1 84.723} C_DIS
LIN {X -0.026,Y -408.857,Z 392.458,A 0.000,B 0.000,C 90.000,E1 82.527} C_DIS
LIN {X -0.055,Y -393.796,Z 392.443,A 0.000,B 0.000,C 90.000,E1 79.746} C_DIS
LIN {X -0.040,Y -383.466,Z 392.432,A 0.000,B 0.000,C 90.000,E1 77.757} C_DIS
LIN {X -0.154,Y -370.428,Z 392.417,A 0.000,B 0.000,C 90.000,E1 75.172} C_DIS
LIN {X 0.059,Y -359.012,Z 392.404,A 0.000,B 0.000,C 90.000,E1 72.779} C_DIS
LIN {X 0.132,Y -346.633,Z 392.389,A 0.000,B 0.000,C 90.000,E1 70.061} C_DIS
LIN {X 0.087,Y -334.583,Z 392.374,A 0.000,B 0.000,C 90.000,E1 67.305} C_DIS
LIN {X -0.156,Y -320.680,Z 392.355,A 0.000,B 0.000,C 90.000,E1 63.896} C_DIS
LIN {X 0.000,Y -307.647,Z 392.335,A 0.000,B 0.000,C 90.000,E1 60.333} C_DIS
LIN {X 0.065,Y -295.572,Z 392.315,A 0.000,B 0.000,C 90.000,E1 56.707} C_DIS
LIN {X 0.005,Y -285.598,Z 392.297,A 0.000,B 0.000,C 90.000,E1 53.371} C_DIS
LIN {X 0.036,Y -278.076,Z 392.281,A 0.000,B 0.000,C 90.000,E1 50.642} C_DIS
LIN {X 0.078,Y -272.494,Z 392.270,A 0.000,B 0.000,C 90.000,E1 48.566} C_DIS
LIN {X -0.030,Y -266.841,Z 392.258,A 0.000,B 0.000,C 90.000,E1 46.500} C_DIS
LIN {X 0.138,Y -260.981,Z 392.247,A 0.000,B 0.000,C 90.000,E1 44.352} C_DIS
LIN {X 0.015,Y -255.051,Z 392.235,A 0.000,B 0.000,C 90.000,E1 42.243} C_DIS
LIN {X -0.026,Y -248.964,Z 392.223,A 0.000,B 0.000,C 90.000,E1 40.092} C_DIS
LIN {X 0.032,Y -240.889,Z 392.206,A 0.000,B 0.000,C 90.000,E1 37.156} C_DIS
LIN {X -0.025,Y -231.326,Z 392.186,A 0.000,B 0.000,C 90.000,E1 33.452} C_DIS
LIN {X -0.047,Y -222.528,Z 392.165,A 0.000,B 0.000,C 90.000,E1 29.667} C_DIS
LIN {X 0.026,Y -216.133,Z 392.148,A 0.000,B 0.000,C 90.000,E1 26.565} C_DIS
LIN {X 0.070,Y -209.051,Z 392.126,A 0.000,B 0.000,C 90.000,E1 22.642} C_DIS
LIN {X 0.075,Y -203.019,Z 392.104,A 0.000,B 0.000,C 90.000,E1 18.671} C_DIS
LIN {X -0.007,Y -198.817,Z 392.086,A 0.000,B 0.000,C 90.000,E1 15.481} C_DIS
LIN {X 0.002,Y -194.426,Z 392.063,A 0.000,B 0.000,C 90.000,E1 11.422} C_DIS
LIN {X -0.079,Y -191.132,Z 392.041,A 0.000,B 0.000,C 90.000,E1 7.352} C_DIS
LIN {X 0.018,Y -188.580,Z 392.009,A 0.000,B 0.000,C 90.000,E1 1.547} C_DIS
LIN {X -0.087,Y -189.899,Z 391.947,A 0.000,B 0.000,C 90.000,E1 350.443} C_DIS
LIN {X 0.019,Y -192.778,Z 391.919,A 0.000,B 0.000,C 90.000,E1 345.463} C_DIS
LIN {X -0.102,Y -196.252,Z 391.897,A 0.000,B 0.000,C 90.000,E1 341.402} C_DIS
LIN {X 0.014,Y -200.864,Z 391.874,A 0.000,B 0.000,C 90.000,E1 337.305} C_DIS
LIN {X -0.064,Y -206.562,Z 391.852,A 0.000,B 0.000,C 90.000,E1 333.307} C_DIS
LIN {X -0.041,Y -213.156,Z 391.830,A 0.000,B 0.000,C 90.000,E1 329.331} C_DIS
LIN {X 0.078,Y -220.511,Z 391.808,A 0.000,B 0.000,C 90.000,E1 325.388} C_DIS
LIN {X 0.027,Y -226.725,Z 391.791,A 0.000,B 0.000,C 90.000,E1 322.316} C_DIS
LIN {X -0.087,Y -233.577,Z 391.774,A 0.000,B 0.000,C 90.000,E1 319.299} C_DIS
LIN {X 0.058,Y -242.260,Z 391.755,A 0.000,B 0.000,C 90.000,E1 315.891} C_DIS
LIN {X -0.047,Y -252.139,Z 391.737,A 0.000,B 0.000,C 90.000,E1 312.609} C_DIS
LIN {X -0.047,Y -261.990,Z 391.721,A 0.000,B 0.000,C 90.000,E1 309.725} C_DIS
LIN {X 0.005,Y -271.220,Z 391.707,A 0.000,B 0.000,C 90.000,E1 307.237} C_DIS
LIN {X -0.055,Y -285.019,Z 391.688,A 0.000,B 0.000,C 90.000,E1 303.785} C_DIS
LIN {X 0.089,Y -299.869,Z 391.669,A 0.000,B 0.000,C 90.000,E1 300.384} C_DIS
LIN {X -0.047,Y -311.474,Z 391.656,A 0.000,B 0.000,C 90.000,E1 298.103} C_DIS
LIN {X -0.001,Y -322.191,Z 391.645,A 0.000,B 0.000,C 90.000,E1 296.155} C_DIS
LIN {X -0.135,Y -331.883,Z 391.636,A 0.000,B 0.000,C 90.000,E1 294.591} C_DIS
LIN {X 0.068,Y -353.263,Z 391.619,A 0.000,B 0.000,C 90.000,E1 291.461} C_DIS
LIN {X 0.003,Y -373.914,Z 391.604,A 0.000,B 0.000,C 90.000,E1 288.779} C_DIS
LIN {X -0.213,Y -391.290,Z 391.593,A 0.000,B 0.000,C 90.000,E1 286.804} C_DIS
LIN {X -0.090,Y -411.770,Z 391.581,A 0.000,B 0.000,C 90.000,E1 284.647} C_DIS
LIN {X 0.056,Y -424.590,Z 391.574,A 0.000,B 0.000,C 90.000,E1 283.355} C_DIS
LIN {X -0.171,Y -434.714,Z 391.569,A 0.000,B 0.000,C 90.000,E1 282.355} C_DIS
LIN {X 0.094,Y -442.052,Z 391.564,A 0.000,B 0.000,C 90.000,E1 281.535} C_DIS
LIN {X -0.209,Y -448.970,Z 391.560,A 0.000,B 0.000,C 90.000,E1 280.782} C_DIS
LIN {X 0.083,Y -455.326,Z 391.555,A 0.000,B 0.000,C 90.000,E1 279.962} C_DIS
LIN {X 0.179,Y -463.020,Z 391.550,A 0.000,B 0.000,C 90.000,E1 278.916} C_DIS
LIN {X -0.164,Y -470.011,Z 391.544,A 0.000,B 0.000,C 90.000,E1 277.936} C_DIS
LIN {X 0.101,Y -476.385,Z 391.538,A 0.000,B 0.000,C 90.000,E1 276.891} C_DIS
LIN {X 0.040,Y -480.651,Z 391.534,A 0.000,B 0.000,C 90.000,E1 276.144} C_DIS
LIN {X 0.071,Y -484.384,Z 391.530,A 0.000,B 0.000,C 90.000,E1 275.391} C_DIS
LIN {X 0.082,Y -487.319,Z 391.526,A 0.000,B 0.000,C 90.000,E1 274.645} C_DIS
LIN {X -0.248,Y -488.778,Z 391.523,A 0.000,B 0.000,C 90.000,E1 274.188} C_DIS
LIN {X -0.045,Y -489.881,Z 391.520,A 0.000,B 0.000,C 90.000,E1 273.669} C_DIS
LIN {X 0.138,Y -490.696,Z 391.518,A 0.000,B 0.000,C 90.000,E1 273.154} C_DIS
LIN {X -0.137,Y -491.218,Z 391.515,A 0.000,B 0.000,C 90.000,E1 272.694} C_DIS
LIN {X 0.060,Y -491.396,Z 391.512,A 0.000,B 0.000,C 90.000,E1 272.178} C_DIS
LIN {X -0.213,Y -491.283,Z 391.509,A 0.000,B 0.000,C 90.000,E1 271.718} C_DIS
LIN {X -0.012,Y -490.772,Z 391.507,A 0.000,B 0.000,C 90.000,E1 271.203} C_DIS
LIN {X 0.190,Y -489.848,Z 391.504,A 0.000,B 0.000,C 90.000,E1 270.688} C_DIS
LIN {X -0.099,Y -488.503,Z 391.501,A 0.000,B 0.000,C 90.000,E1 270.229} C_DIS
LIN {X 0.095,Y -486.590,Z 391.498,A 0.000,B 0.000,C 90.000,E1 269.714} C_DIS
LIN {X -0.205,Y -483.987,Z 391.496,A 0.000,B 0.000,C 90.000,E1 269.255} C_DIS
LIN {X 0.120,Y -482.435,Z 391.494,A 0.000,B 0.000,C 90.000,E1 268.969} C_DIS
LIN {X -0.204,Y -478.599,Z 391.492,A 0.000,B 0.000,C 90.000,E1 268.511} C_DIS
LIN {X -0.052,Y -473.618,Z 391.489,A 0.000,B 0.000,C 90.000,E1 267.993} C_DIS
LIN {X -0.225,Y -470.673,Z 391.487,A 0.000,B 0.000,C 90.000,E1 267.764} C_DIS
LIN {X -0.119,Y -464.234,Z 391.485,A 0.000,B 0.000,C 90.000,E1 267.306} C_DIS
LIN {X 0.084,Y -457.228,Z 391.483,A 0.000,B 0.000,C 90.000,E1 266.906} C_DIS
LIN {X 0.003,Y -450.105,Z 391.481,A 0.000,B 0.000,C 90.000,E1 266.617} C_DIS
LIN {X -0.092,Y -442.887,Z 391.480,A 0.000,B 0.000,C 90.000,E1 266.388} C_DIS
LIN {X 0.149,Y -434.764,Z 391.479,A 0.000,B 0.000,C 90.000,E1 266.159} C_DIS
LIN {X -0.031,Y -426.742,Z 391.478,A 0.000,B 0.000,C 90.000,E1 266.045} C_DIS
LIN {X -0.184,Y -419.712,Z 391.478,A 0.000,B 0.000,C 90.000,E1 265.988} C_DIS
LIN {X -0.035,Y -410.495,Z 391.477,A 0.000,B 0.000,C 90.000,E1 265.927} C_DIS
LIN {X -0.039,Y -180.917,Z 391.477,A 0.000,B 0.000,C 90.000,E1 265.927} C_DIS
LIN {X 0.083,Y -180.869,Z 391.472,A 0.000,B 0.000,C 90.000,E1 265.008} C_DIS
LIN {X -0.040,Y -178.985,Z 391.444,A 0.000,B 0.000,C 90.000,E1 259.982} C_DIS
LIN {X -0.029,Y -177.961,Z 391.435,A 0.000,B 0.000,C 90.000,E1 258.285} C_DIS
LIN {X -0.010,Y -175.603,Z 391.411,A 0.000,B 0.000,C 90.000,E1 254.031} C_DIS
LIN {X 0.002,Y -172.327,Z 391.388,A 0.000,B 0.000,C 90.000,E1 249.752} C_DIS
LIN {X -0.019,Y -171.804,Z 391.383,A 0.000,B 0.000,C 90.000,E1 248.901} C_DIS
LIN {X 0.019,Y -169.479,Z 391.368,A 0.000,B 0.000,C 90.000,E1 246.305} C_DIS
LIN {X -0.074,Y -166.805,Z 391.349,A 0.000,B 0.000,C 90.000,E1 242.871} C_DIS
LIN {X 0.069,Y -162.787,Z 391.325,A 0.000,B 0.000,C 90.000,E1 238.456} C_DIS
LIN {X 0.044,Y -161.475,Z 391.315,A 0.000,B 0.000,C 90.000,E1 236.707} C_DIS
LIN {X 0.085,Y -157.470,Z 391.291,A 0.000,B 0.000,C 90.000,E1 232.271} C_DIS
LIN {X 0.017,Y -155.485,Z 391.276,A 0.000,B 0.000,C 90.000,E1 229.622} C_DIS
LIN {X -0.050,Y -151.793,Z 391.251,A 0.000,B 0.000,C 90.000,E1 225.162} C_DIS
LIN {X -0.037,Y -150.001,Z 391.236,A 0.000,B 0.000,C 90.000,E1 222.447} C_DIS
LIN {X -0.006,Y -146.829,Z 391.210,A 0.000,B 0.000,C 90.000,E1 217.890} C_DIS
LIN {X -0.019,Y -145.410,Z 391.195,A 0.000,B 0.000,C 90.000,E1 215.152} C_DIS
LIN {X 0.016,Y -142.840,Z 391.170,A 0.000,B 0.000,C 90.000,E1 210.541} C_DIS
LIN {X -0.054,Y -141.454,Z 391.149,A 0.000,B 0.000,C 90.000,E1 206.873} C_DIS
LIN {X -0.013,Y -139.372,Z 391.113,A 0.000,B 0.000,C 90.000,E1 200.355} C_DIS
LIN {X -0.072,Y -138.822,Z 391.098,A 0.000,B 0.000,C 90.000,E1 197.583} C_DIS
LIN {X 0.017,Y -138.352,Z 391.056,A 0.000,B 0.000,C 90.000,E1 190.074} C_DIS
LIN {X -0.010,Y -139.533,Z 391.004,A 0.000,B 0.000,C 90.000,E1 180.745} C_DIS
LIN {X -0.058,Y -141.215,Z 390.973,A 0.000,B 0.000,C 90.000,E1 175.179} C_DIS
LIN {X 0.043,Y -142.588,Z 390.958,A 0.000,B 0.000,C 90.000,E1 172.356} C_DIS
